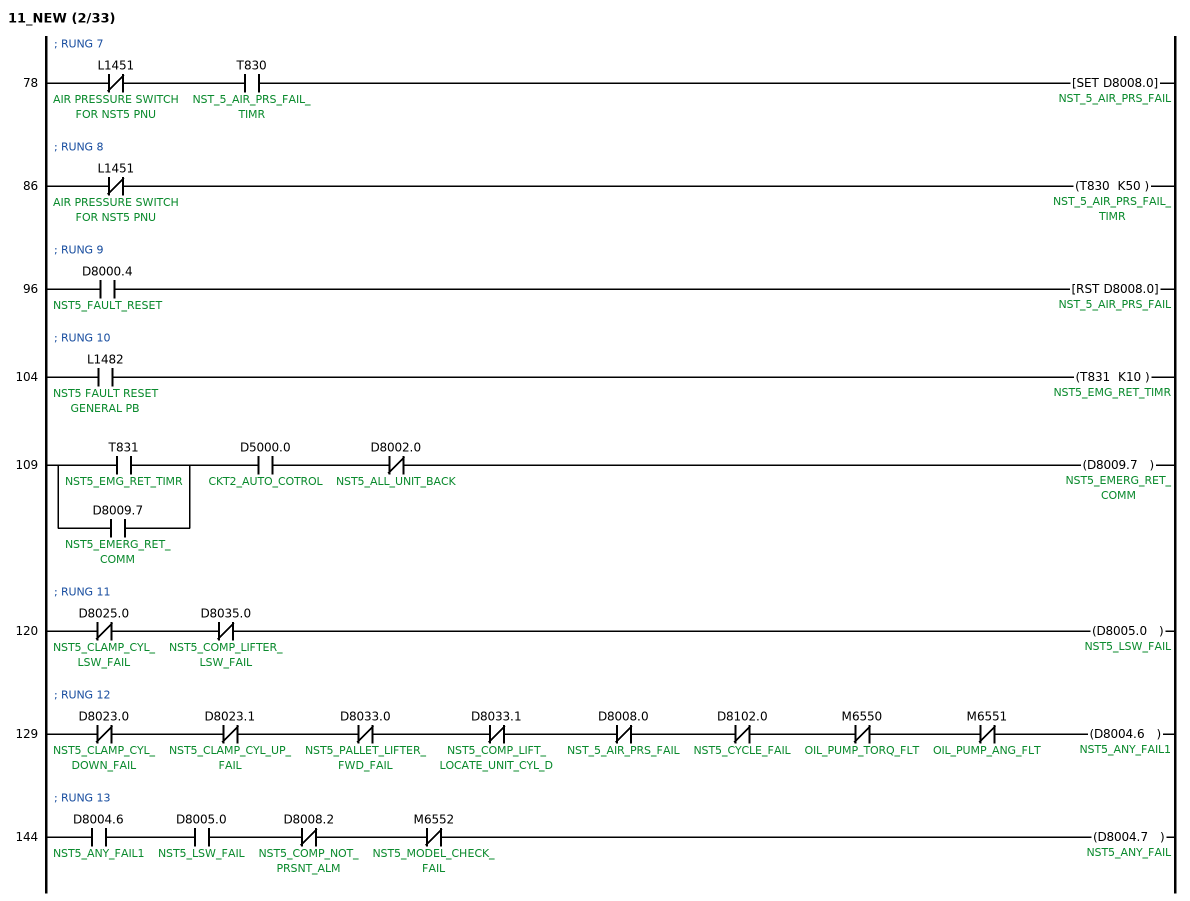
[picture p192: ladder of 11_NEW, rungs at steps 78 to 144]
; RUNG 7
78    LDI     L1451  ; AIR PRESSURE SWITCH FOR NST5 PNU
      AND     T830  ; NST_5_AIR_PRS_FAIL_TIMR
      SET     D8008.0  ; NST_5_AIR_PRS_FAIL
; RUNG 8
86    LDI     L1451  ; AIR PRESSURE SWITCH FOR NST5 PNU
      OUT     T830 K50  ; NST_5_AIR_PRS_FAIL_TIMR
; RUNG 9
96    LD      D8000.4  ; NST5_FAULT_RESET
      RST     D8008.0  ; NST_5_AIR_PRS_FAIL
; RUNG 10
104   LD      L1482  ; NST5 FAULT RESET GENERAL PB
      OUT     T831 K10  ; NST5_EMG_RET_TIMR
109   LD      T831  ; NST5_EMG_RET_TIMR
      OR      D8009.7  ; NST5_EMERG_RET_COMM
      AND     D5000.0  ; CKT2_AUTO_COTROL
      ANI     D8002.0  ; NST5_ALL_UNIT_BACK
      OUT     D8009.7  ; NST5_EMERG_RET_COMM
; RUNG 11
120   LDI     D8025.0  ; NST5_CLAMP_CYL_LSW_FAIL
      ANI     D8035.0  ; NST5_COMP_LIFTER_LSW_FAIL
      OUT     D8005.0  ; NST5_LSW_FAIL
; RUNG 12
129   LDI     D8023.0  ; NST5_CLAMP_CYL_DOWN_FAIL
      ANI     D8023.1  ; NST5_CLAMP_CYL_UP_FAIL
      ANI     D8033.0  ; NST5_PALLET_LIFTER_FWD_FAIL
      ANI     D8033.1  ; NST5_COMP_LIFT_LOCATE_UNIT_CYL_D
      ANI     D8008.0  ; NST_5_AIR_PRS_FAIL
      ANI     D8102.0  ; NST5_CYCLE_FAIL
      ANI     M6550  ; OIL_PUMP_TORQ_FLT
      ANI     M6551  ; OIL_PUMP_ANG_FLT
      OUT     D8004.6  ; NST5_ANY_FAIL1
; RUNG 13
144   LD      D8004.6  ; NST5_ANY_FAIL1
      AND     D8005.0  ; NST5_LSW_FAIL
      ANI     D8008.2  ; NST5_COMP_NOT_PRSNT_ALM
      ANI     M6552  ; NST5_MODEL_CHECK_FAIL
      OUT     D8004.7  ; NST5_ANY_FAIL
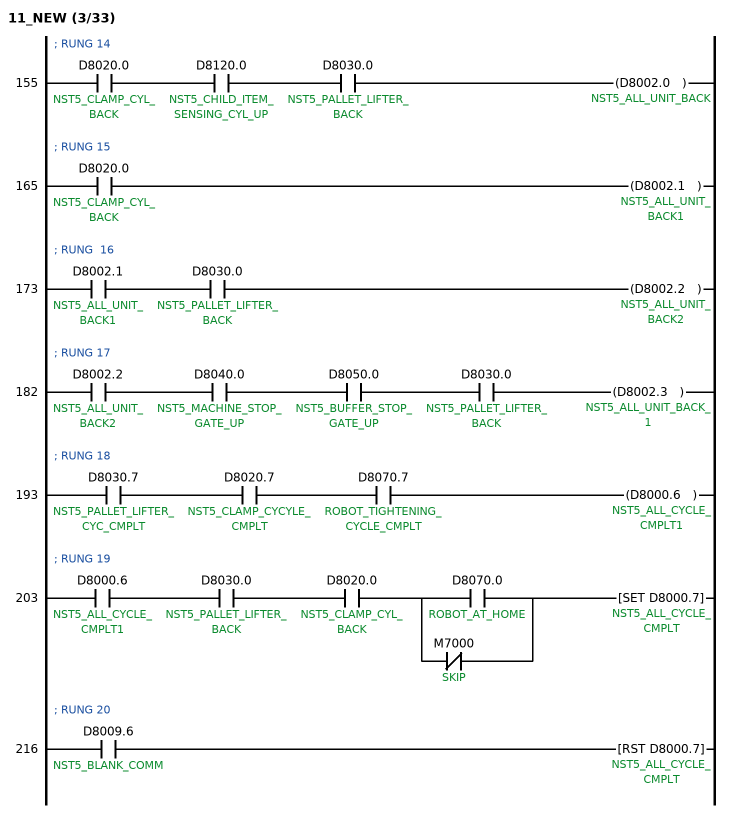
; RUNG 14
155   LD      D8020.0  ; NST5_CLAMP_CYL_BACK
      AND     D8120.0  ; NST5_CHILD_ITEM_SENSING_CYL_UP
      AND     D8030.0  ; NST5_PALLET_LIFTER_BACK
      OUT     D8002.0  ; NST5_ALL_UNIT_BACK
; RUNG 15
165   LD      D8020.0  ; NST5_CLAMP_CYL_BACK
      OUT     D8002.1  ; NST5_ALL_UNIT_BACK1
; RUNG  16
173   LD      D8002.1  ; NST5_ALL_UNIT_BACK1
      AND     D8030.0  ; NST5_PALLET_LIFTER_BACK
      OUT     D8002.2  ; NST5_ALL_UNIT_BACK2
; RUNG 17
182   LD      D8002.2  ; NST5_ALL_UNIT_BACK2
      AND     D8040.0  ; NST5_MACHINE_STOP_GATE_UP
      AND     D8050.0  ; NST5_BUFFER_STOP_GATE_UP
      AND     D8030.0  ; NST5_PALLET_LIFTER_BACK
      OUT     D8002.3  ; NST5_ALL_UNIT_BACK_1
; RUNG 18
193   LD      D8030.7  ; NST5_PALLET_LIFTER_CYC_CMPLT
      AND     D8020.7  ; NST5_CLAMP_CYCYLE_CMPLT
      AND     D8070.7  ; ROBOT_TIGHTENING_CYCLE_CMPLT
      OUT     D8000.6  ; NST5_ALL_CYCLE_CMPLT1
; RUNG 19
203   LD      D8000.6  ; NST5_ALL_CYCLE_CMPLT1
      AND     D8030.0  ; NST5_PALLET_LIFTER_BACK
      AND     D8020.0  ; NST5_CLAMP_CYL_BACK
      LD      D8070.0  ; ROBOT_AT_HOME
      ORI     M7000  ; SKIP
      ANB
      SET     D8000.7  ; NST5_ALL_CYCLE_CMPLT
; RUNG 20
216   LD      D8009.6  ; NST5_BLANK_COMM
      RST     D8000.7  ; NST5_ALL_CYCLE_CMPLT
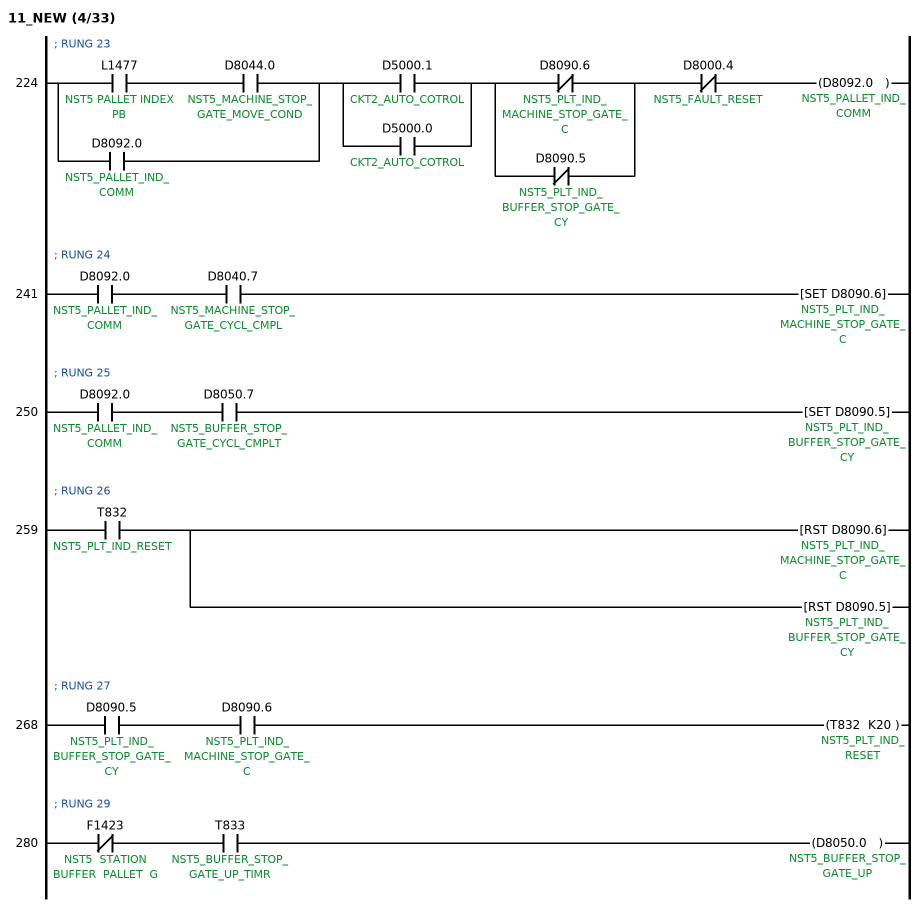
; RUNG 23
224   LD      L1477  ; NST5 PALLET INDEX PB
      AND     D8044.0  ; NST5_MACHINE_STOP_GATE_MOVE_COND
      OR      D8092.0  ; NST5_PALLET_IND_COMM
      LD      D5000.1  ; CKT2_AUTO_COTROL
      OR      D5000.0  ; CKT2_AUTO_COTROL
      ANB
      LDI     D8090.6  ; NST5_PLT_IND_MACHINE_STOP_GATE_C
      ORI     D8090.5  ; NST5_PLT_IND_BUFFER_STOP_GATE_CY
      ANB
      ANI     D8000.4  ; NST5_FAULT_RESET
      OUT     D8092.0  ; NST5_PALLET_IND_COMM
; RUNG 24
241   LD      D8092.0  ; NST5_PALLET_IND_COMM
      AND     D8040.7  ; NST5_MACHINE_STOP_GATE_CYCL_CMPL
      SET     D8090.6  ; NST5_PLT_IND_MACHINE_STOP_GATE_C
; RUNG 25
250   LD      D8092.0  ; NST5_PALLET_IND_COMM
      AND     D8050.7  ; NST5_BUFFER_STOP_GATE_CYCL_CMPLT
      SET     D8090.5  ; NST5_PLT_IND_BUFFER_STOP_GATE_CY
; RUNG 26
259   LD      T832  ; NST5_PLT_IND_RESET
      RST     D8090.6  ; NST5_PLT_IND_MACHINE_STOP_GATE_C
      RST     D8090.5  ; NST5_PLT_IND_BUFFER_STOP_GATE_CY
; RUNG 27
268   LD      D8090.5  ; NST5_PLT_IND_BUFFER_STOP_GATE_CY
      AND     D8090.6  ; NST5_PLT_IND_MACHINE_STOP_GATE_C
      OUT     T832 K20  ; NST5_PLT_IND_RESET
; RUNG 29
280   LDI     F1423  ; NST5  STATION  BUFFER  PALLET  G
      AND     T833  ; NST5_BUFFER_STOP_GATE_UP_TIMR
      OUT     D8050.0  ; NST5_BUFFER_STOP_GATE_UP
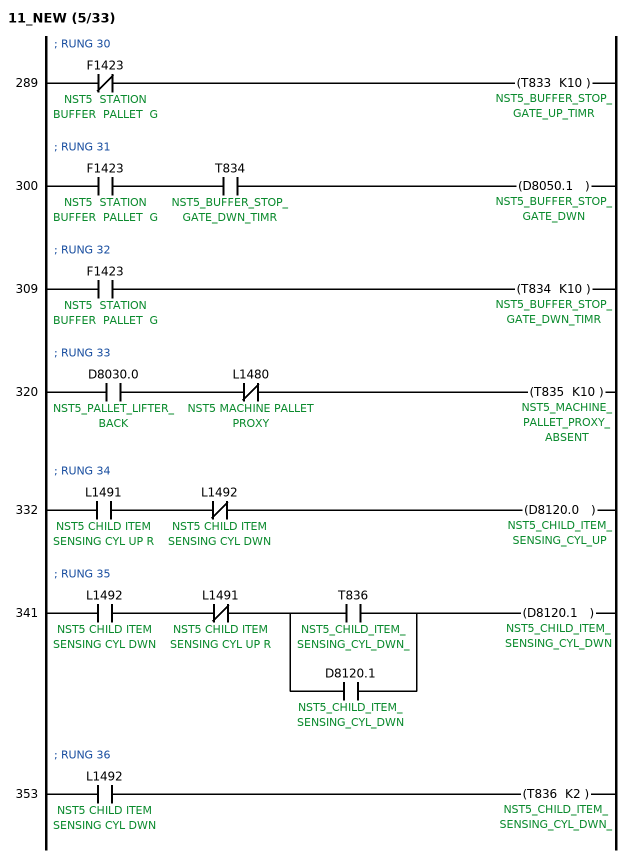
; RUNG 30
289   LDI     F1423  ; NST5  STATION  BUFFER  PALLET  G
      OUT     T833 K10  ; NST5_BUFFER_STOP_GATE_UP_TIMR
; RUNG 31
300   LD      F1423  ; NST5  STATION  BUFFER  PALLET  G
      AND     T834  ; NST5_BUFFER_STOP_GATE_DWN_TIMR
      OUT     D8050.1  ; NST5_BUFFER_STOP_GATE_DWN
; RUNG 32
309   LD      F1423  ; NST5  STATION  BUFFER  PALLET  G
      OUT     T834 K10  ; NST5_BUFFER_STOP_GATE_DWN_TIMR
; RUNG 33
320   LD      D8030.0  ; NST5_PALLET_LIFTER_BACK
      ANI     L1480  ; NST5 MACHINE PALLET PROXY
      OUT     T835 K10  ; NST5_MACHINE_PALLET_PROXY_ABSENT
; RUNG 34
332   LD      L1491  ; NST5 CHILD ITEM SENSING CYL UP R
      ANI     L1492  ; NST5 CHILD ITEM SENSING CYL DWN
      OUT     D8120.0  ; NST5_CHILD_ITEM_SENSING_CYL_UP
; RUNG 35
341   LD      L1492  ; NST5 CHILD ITEM SENSING CYL DWN
      ANI     L1491  ; NST5 CHILD ITEM SENSING CYL UP R
      LD      T836  ; NST5_CHILD_ITEM_SENSING_CYL_DWN_
      OR      D8120.1  ; NST5_CHILD_ITEM_SENSING_CYL_DWN
      ANB
      OUT     D8120.1  ; NST5_CHILD_ITEM_SENSING_CYL_DWN
; RUNG 36
353   LD      L1492  ; NST5 CHILD ITEM SENSING CYL DWN
      OUT     T836 K2  ; NST5_CHILD_ITEM_SENSING_CYL_DWN_
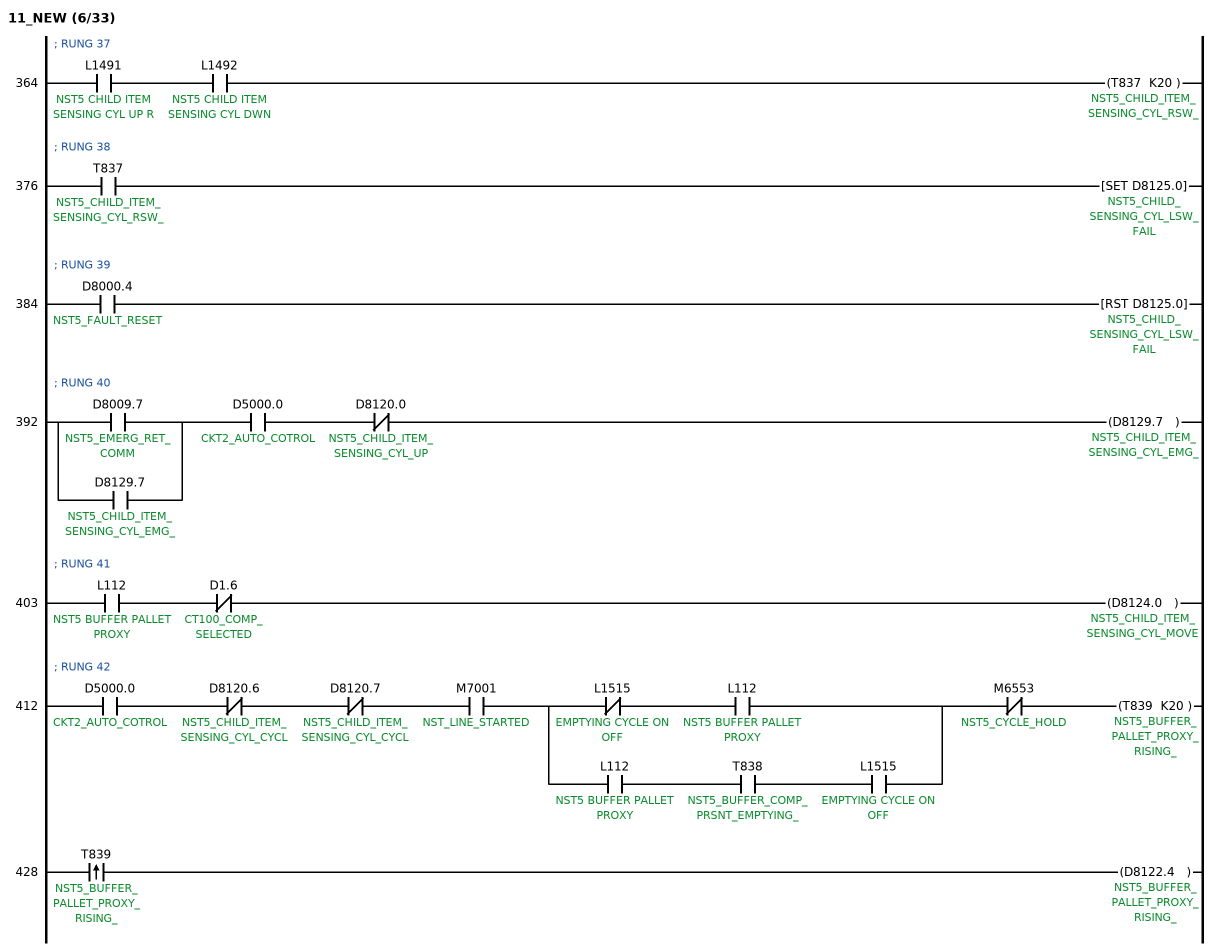
; RUNG 37
364   LD      L1491  ; NST5 CHILD ITEM SENSING CYL UP R
      AND     L1492  ; NST5 CHILD ITEM SENSING CYL DWN
      OUT     T837 K20  ; NST5_CHILD_ITEM_SENSING_CYL_RSW_
; RUNG 38
376   LD      T837  ; NST5_CHILD_ITEM_SENSING_CYL_RSW_
      SET     D8125.0  ; NST5_CHILD_SENSING_CYL_LSW_FAIL
; RUNG 39
384   LD      D8000.4  ; NST5_FAULT_RESET
      RST     D8125.0  ; NST5_CHILD_SENSING_CYL_LSW_FAIL
; RUNG 40
392   LD      D8009.7  ; NST5_EMERG_RET_COMM
      OR      D8129.7  ; NST5_CHILD_ITEM_SENSING_CYL_EMG_
      AND     D5000.0  ; CKT2_AUTO_COTROL
      ANI     D8120.0  ; NST5_CHILD_ITEM_SENSING_CYL_UP
      OUT     D8129.7  ; NST5_CHILD_ITEM_SENSING_CYL_EMG_
; RUNG 41
403   LD      L112  ; NST5 BUFFER PALLET PROXY
      ANI     D1.6  ; CT100_COMP_SELECTED
      OUT     D8124.0  ; NST5_CHILD_ITEM_SENSING_CYL_MOVE
; RUNG 42
412   LD      D5000.0  ; CKT2_AUTO_COTROL
      ANI     D8120.6  ; NST5_CHILD_ITEM_SENSING_CYL_CYCL
      ANI     D8120.7  ; NST5_CHILD_ITEM_SENSING_CYL_CYCL
      AND     M7001  ; NST_LINE_STARTED
      LDI     L1515  ; EMPTYING CYCLE ON OFF
      AND     L112  ; NST5 BUFFER PALLET PROXY
      LD      L112  ; NST5 BUFFER PALLET PROXY
      AND     T838  ; NST5_BUFFER_COMP_PRSNT_EMPTYING_
      AND     L1515  ; EMPTYING CYCLE ON OFF
      ORB
      ANB
      ANI     M6553  ; NST5_CYCLE_HOLD
      OUT     T839 K20  ; NST5_BUFFER_PALLET_PROXY_RISING_
428   LDP     T839  ; NST5_BUFFER_PALLET_PROXY_RISING_
      OUT     D8122.4  ; NST5_BUFFER_PALLET_PROXY_RISING_
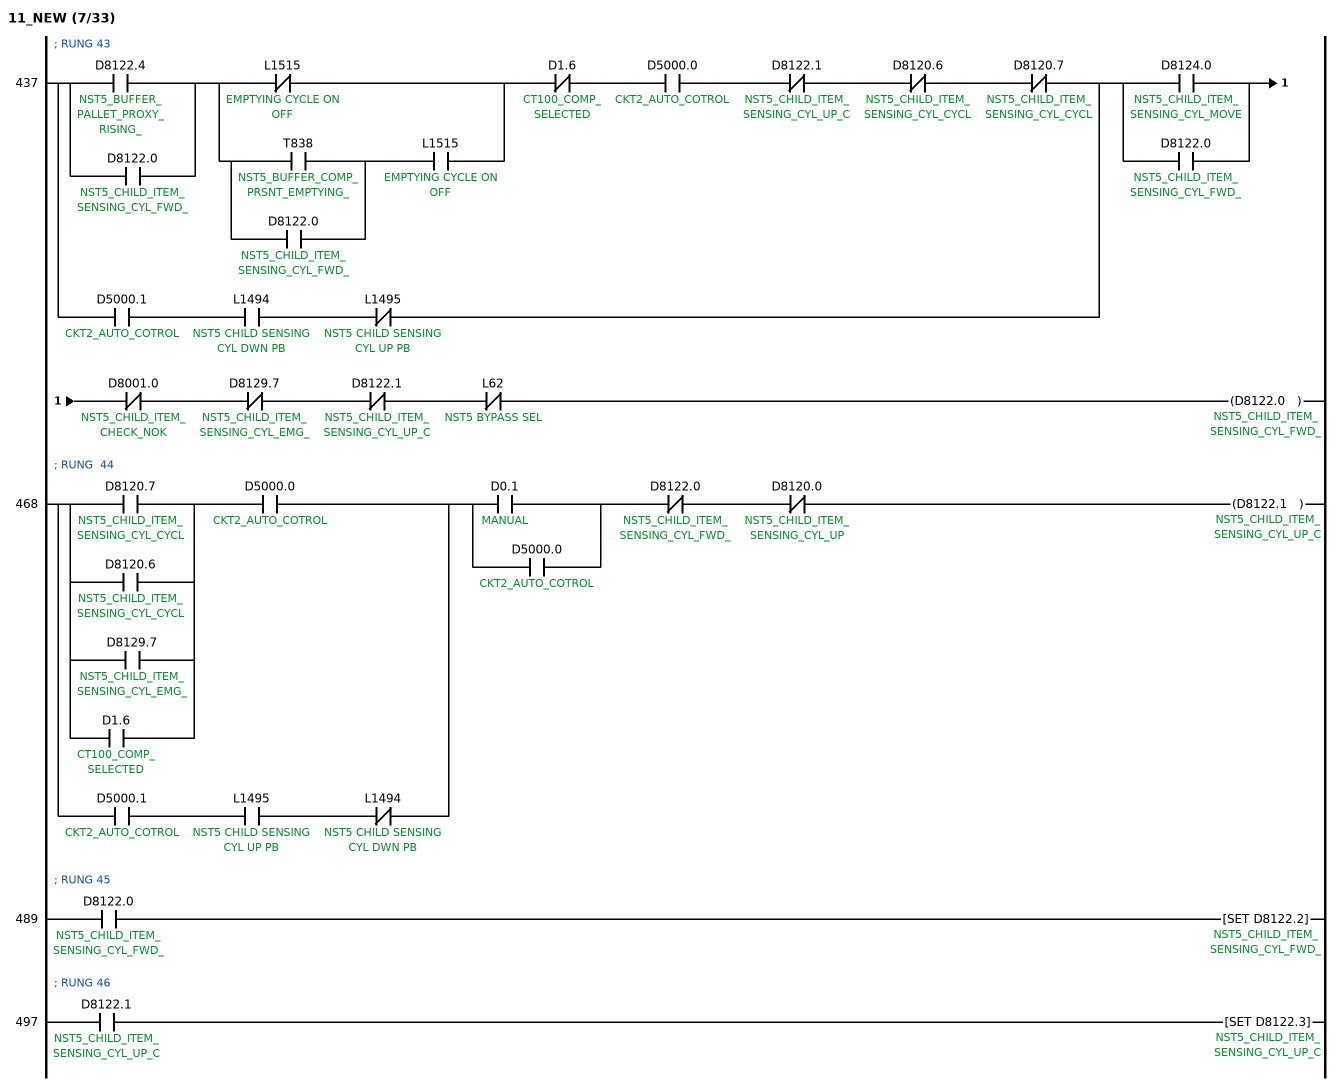
; RUNG 43
437   LD      D8122.4  ; NST5_BUFFER_PALLET_PROXY_RISING_
      OR      D8122.0  ; NST5_CHILD_ITEM_SENSING_CYL_FWD_
      LDI     L1515  ; EMPTYING CYCLE ON OFF
      LD      T838  ; NST5_BUFFER_COMP_PRSNT_EMPTYING_
      OR      D8122.0  ; NST5_CHILD_ITEM_SENSING_CYL_FWD_
      AND     L1515  ; EMPTYING CYCLE ON OFF
      ORB
      ANB
      ANI     D1.6  ; CT100_COMP_SELECTED
      AND     D5000.0  ; CKT2_AUTO_COTROL
      ANI     D8122.1  ; NST5_CHILD_ITEM_SENSING_CYL_UP_C
      ANI     D8120.6  ; NST5_CHILD_ITEM_SENSING_CYL_CYCL
      ANI     D8120.7  ; NST5_CHILD_ITEM_SENSING_CYL_CYCL
      LD      D5000.1  ; CKT2_AUTO_COTROL
      AND     L1494  ; NST5 CHILD SENSING CYL DWN PB
      ANI     L1495  ; NST5 CHILD SENSING CYL UP PB
      ORB
      LD      D8124.0  ; NST5_CHILD_ITEM_SENSING_CYL_MOVE
      OR      D8122.0  ; NST5_CHILD_ITEM_SENSING_CYL_FWD_
      ANB
      ANI     D8001.0  ; NST5_CHILD_ITEM_CHECK_NOK
      ANI     D8129.7  ; NST5_CHILD_ITEM_SENSING_CYL_EMG_
      ANI     D8122.1  ; NST5_CHILD_ITEM_SENSING_CYL_UP_C
      ANI     L62  ; NST5 BYPASS SEL
      OUT     D8122.0  ; NST5_CHILD_ITEM_SENSING_CYL_FWD_
; RUNG  44
468   LD      D8120.7  ; NST5_CHILD_ITEM_SENSING_CYL_CYCL
      OR      D8120.6  ; NST5_CHILD_ITEM_SENSING_CYL_CYCL
      OR      D8129.7  ; NST5_CHILD_ITEM_SENSING_CYL_EMG_
      OR      D1.6  ; CT100_COMP_SELECTED
      AND     D5000.0  ; CKT2_AUTO_COTROL
      LD      D5000.1  ; CKT2_AUTO_COTROL
      AND     L1495  ; NST5 CHILD SENSING CYL UP PB
      ANI     L1494  ; NST5 CHILD SENSING CYL DWN PB
      ORB
      LD      D0.1  ; MANUAL
      OR      D5000.0  ; CKT2_AUTO_COTROL
      ANB
      ANI     D8122.0  ; NST5_CHILD_ITEM_SENSING_CYL_FWD_
      ANI     D8120.0  ; NST5_CHILD_ITEM_SENSING_CYL_UP
      OUT     D8122.1  ; NST5_CHILD_ITEM_SENSING_CYL_UP_C
; RUNG 45
489   LD      D8122.0  ; NST5_CHILD_ITEM_SENSING_CYL_FWD_
      SET     D8122.2  ; NST5_CHILD_ITEM_SENSING_CYL_FWD_
; RUNG 46
497   LD      D8122.1  ; NST5_CHILD_ITEM_SENSING_CYL_UP_C
      SET     D8122.3  ; NST5_CHILD_ITEM_SENSING_CYL_UP_C
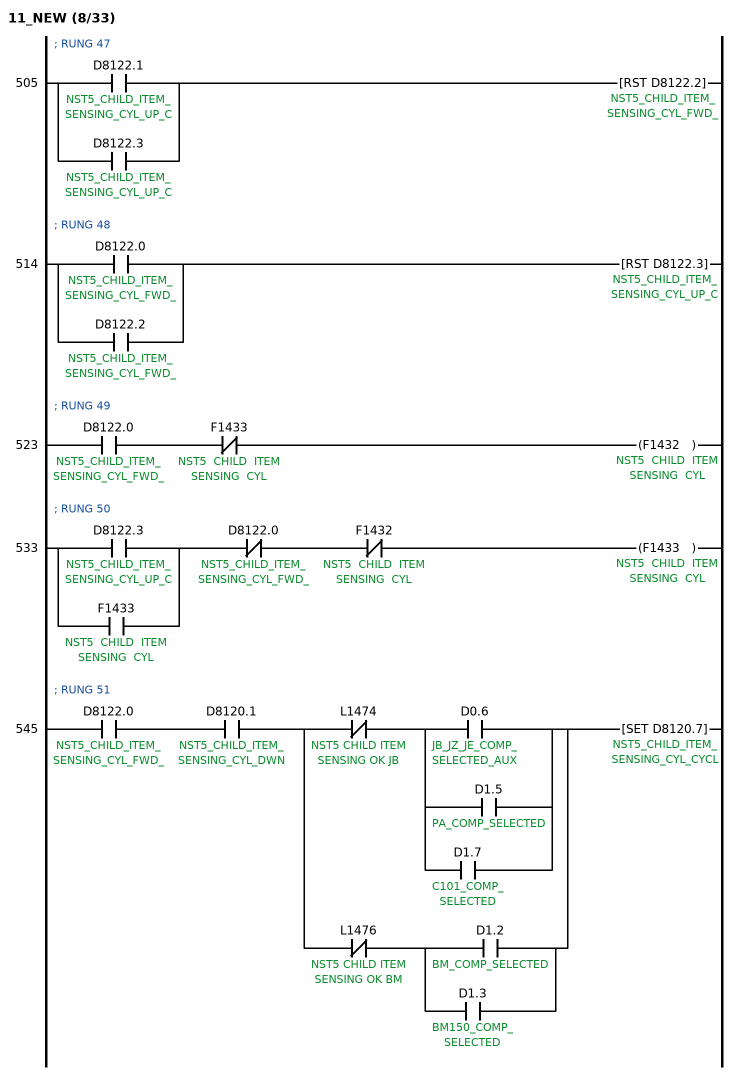
; RUNG 47
505   LD      D8122.1  ; NST5_CHILD_ITEM_SENSING_CYL_UP_C
      OR      D8122.3  ; NST5_CHILD_ITEM_SENSING_CYL_UP_C
      RST     D8122.2  ; NST5_CHILD_ITEM_SENSING_CYL_FWD_
; RUNG 48
514   LD      D8122.0  ; NST5_CHILD_ITEM_SENSING_CYL_FWD_
      OR      D8122.2  ; NST5_CHILD_ITEM_SENSING_CYL_FWD_
      RST     D8122.3  ; NST5_CHILD_ITEM_SENSING_CYL_UP_C
; RUNG 49
523   LD      D8122.0  ; NST5_CHILD_ITEM_SENSING_CYL_FWD_
      ANI     F1433  ; NST5  CHILD  ITEM  SENSING  CYL
      OUT     F1432  ; NST5  CHILD  ITEM  SENSING  CYL
; RUNG 50
533   LD      D8122.3  ; NST5_CHILD_ITEM_SENSING_CYL_UP_C
      OR      F1433  ; NST5  CHILD  ITEM  SENSING  CYL
      ANI     D8122.0  ; NST5_CHILD_ITEM_SENSING_CYL_FWD_
      ANI     F1432  ; NST5  CHILD  ITEM  SENSING  CYL
      OUT     F1433  ; NST5  CHILD  ITEM  SENSING  CYL
; RUNG 51
545   LD      D8122.0  ; NST5_CHILD_ITEM_SENSING_CYL_FWD_
      AND     D8120.1  ; NST5_CHILD_ITEM_SENSING_CYL_DWN
      LDI     L1474  ; NST5 CHILD ITEM SENSING OK JB
      LD      D0.6  ; JB_JZ_JE_COMP_SELECTED_AUX
      OR      D1.5  ; PA_COMP_SELECTED
      OR      D1.7  ; C101_COMP_SELECTED
      ANB
      LDI     L1476  ; NST5 CHILD ITEM SENSING OK BM
      LD      D1.2  ; BM_COMP_SELECTED
      OR      D1.3  ; BM150_COMP_SELECTED
      ANB
      ORB
      ANB
      SET     D8120.7  ; NST5_CHILD_ITEM_SENSING_CYL_CYCL
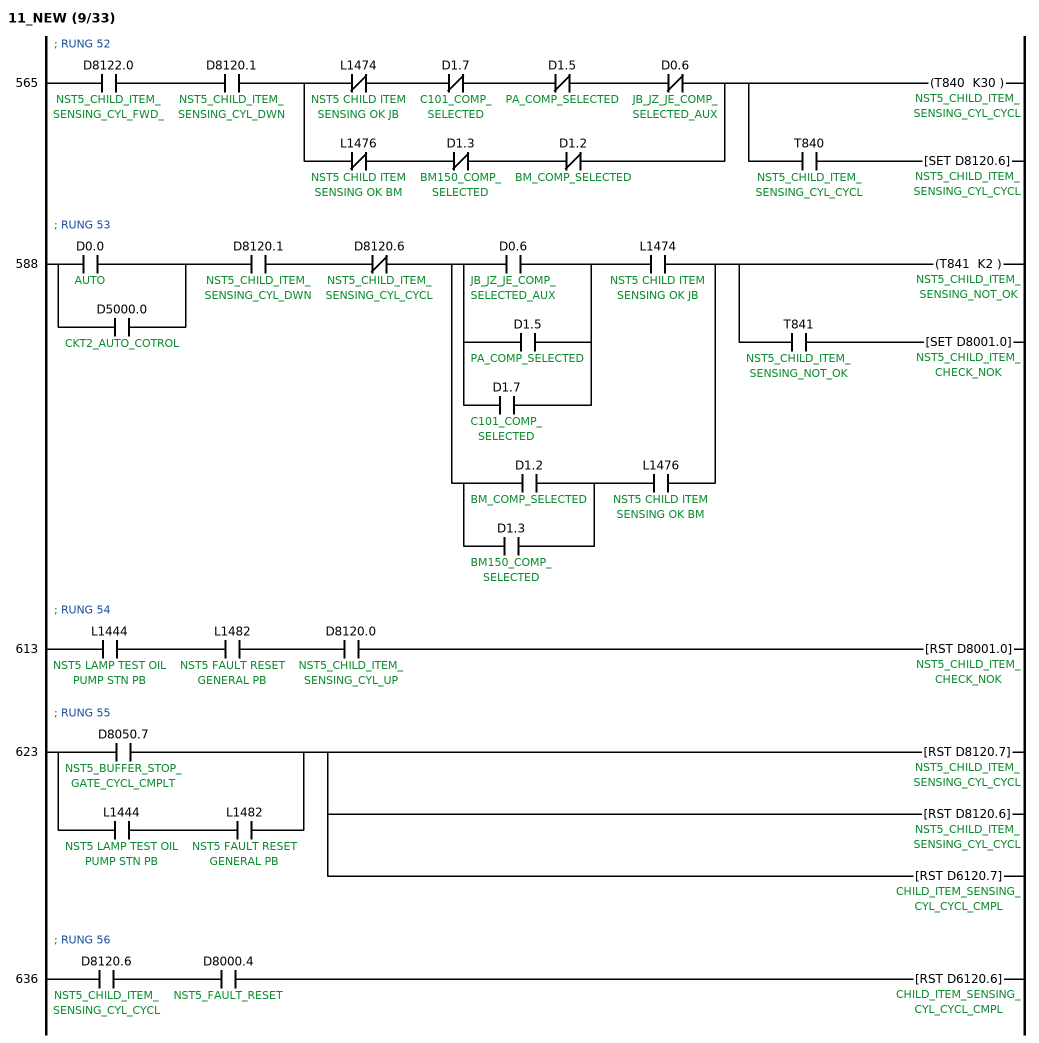
; RUNG 52
565   LD      D8122.0  ; NST5_CHILD_ITEM_SENSING_CYL_FWD_
      AND     D8120.1  ; NST5_CHILD_ITEM_SENSING_CYL_DWN
      LDI     L1474  ; NST5 CHILD ITEM SENSING OK JB
      ANI     D1.7  ; C101_COMP_SELECTED
      ANI     D1.5  ; PA_COMP_SELECTED
      ANI     D0.6  ; JB_JZ_JE_COMP_SELECTED_AUX
      LDI     L1476  ; NST5 CHILD ITEM SENSING OK BM
      ANI     D1.3  ; BM150_COMP_SELECTED
      ANI     D1.2  ; BM_COMP_SELECTED
      ORB
      ANB
      OUT     T840 K30  ; NST5_CHILD_ITEM_SENSING_CYL_CYCL
      AND     T840  ; NST5_CHILD_ITEM_SENSING_CYL_CYCL
      SET     D8120.6  ; NST5_CHILD_ITEM_SENSING_CYL_CYCL
; RUNG 53
588   LD      D0.0  ; AUTO
      OR      D5000.0  ; CKT2_AUTO_COTROL
      AND     D8120.1  ; NST5_CHILD_ITEM_SENSING_CYL_DWN
      ANI     D8120.6  ; NST5_CHILD_ITEM_SENSING_CYL_CYCL
      LD      D0.6  ; JB_JZ_JE_COMP_SELECTED_AUX
      OR      D1.5  ; PA_COMP_SELECTED
      OR      D1.7  ; C101_COMP_SELECTED
      AND     L1474  ; NST5 CHILD ITEM SENSING OK JB
      LD      D1.2  ; BM_COMP_SELECTED
      OR      D1.3  ; BM150_COMP_SELECTED
      AND     L1476  ; NST5 CHILD ITEM SENSING OK BM
      ORB
      ANB
      OUT     T841 K2  ; NST5_CHILD_ITEM_SENSING_NOT_OK
      AND     T841  ; NST5_CHILD_ITEM_SENSING_NOT_OK
      SET     D8001.0  ; NST5_CHILD_ITEM_CHECK_NOK
; RUNG 54
613   LD      L1444  ; NST5 LAMP TEST OIL PUMP STN PB
      AND     L1482  ; NST5 FAULT RESET GENERAL PB
      AND     D8120.0  ; NST5_CHILD_ITEM_SENSING_CYL_UP
      RST     D8001.0  ; NST5_CHILD_ITEM_CHECK_NOK
; RUNG 55
623   LD      D8050.7  ; NST5_BUFFER_STOP_GATE_CYCL_CMPLT
      LD      L1444  ; NST5 LAMP TEST OIL PUMP STN PB
      AND     L1482  ; NST5 FAULT RESET GENERAL PB
      ORB
      RST     D8120.7  ; NST5_CHILD_ITEM_SENSING_CYL_CYCL
      RST     D8120.6  ; NST5_CHILD_ITEM_SENSING_CYL_CYCL
      RST     D6120.7  ; CHILD_ITEM_SENSING_CYL_CYCL_CMPL
; RUNG 56
636   LD      D8120.6  ; NST5_CHILD_ITEM_SENSING_CYL_CYCL
      AND     D8000.4  ; NST5_FAULT_RESET
      RST     D6120.6  ; CHILD_ITEM_SENSING_CYL_CYCL_CMPL
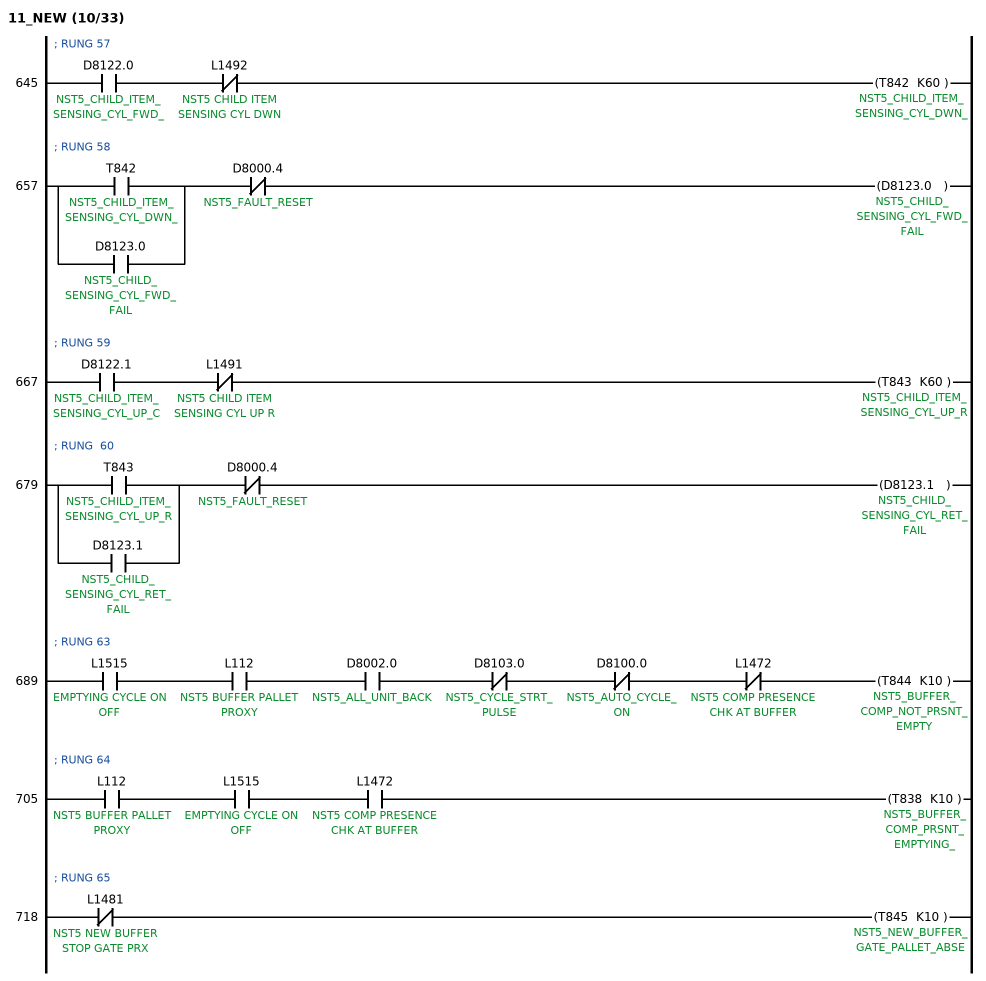
; RUNG 57
645   LD      D8122.0  ; NST5_CHILD_ITEM_SENSING_CYL_FWD_
      ANI     L1492  ; NST5 CHILD ITEM SENSING CYL DWN
      OUT     T842 K60  ; NST5_CHILD_ITEM_SENSING_CYL_DWN_
; RUNG 58
657   LD      T842  ; NST5_CHILD_ITEM_SENSING_CYL_DWN_
      OR      D8123.0  ; NST5_CHILD_SENSING_CYL_FWD_FAIL
      ANI     D8000.4  ; NST5_FAULT_RESET
      OUT     D8123.0  ; NST5_CHILD_SENSING_CYL_FWD_FAIL
; RUNG 59
667   LD      D8122.1  ; NST5_CHILD_ITEM_SENSING_CYL_UP_C
      ANI     L1491  ; NST5 CHILD ITEM SENSING CYL UP R
      OUT     T843 K60  ; NST5_CHILD_ITEM_SENSING_CYL_UP_R
; RUNG  60
679   LD      T843  ; NST5_CHILD_ITEM_SENSING_CYL_UP_R
      OR      D8123.1  ; NST5_CHILD_SENSING_CYL_RET_FAIL
      ANI     D8000.4  ; NST5_FAULT_RESET
      OUT     D8123.1  ; NST5_CHILD_SENSING_CYL_RET_FAIL
; RUNG 63
689   LD      L1515  ; EMPTYING CYCLE ON OFF
      AND     L112  ; NST5 BUFFER PALLET PROXY
      AND     D8002.0  ; NST5_ALL_UNIT_BACK
      ANI     D8103.0  ; NST5_CYCLE_STRT_PULSE
      ANI     D8100.0  ; NST5_AUTO_CYCLE_ON
      ANI     L1472  ; NST5 COMP PRESENCE CHK AT BUFFER
      OUT     T844 K10  ; NST5_BUFFER_COMP_NOT_PRSNT_EMPTY
; RUNG 64
705   LD      L112  ; NST5 BUFFER PALLET PROXY
      AND     L1515  ; EMPTYING CYCLE ON OFF
      AND     L1472  ; NST5 COMP PRESENCE CHK AT BUFFER
      OUT     T838 K10  ; NST5_BUFFER_COMP_PRSNT_EMPTYING_
; RUNG 65
718   LDI     L1481  ; NST5 NEW BUFFER STOP GATE PRX
      OUT     T845 K10  ; NST5_NEW_BUFFER_GATE_PALLET_ABSE
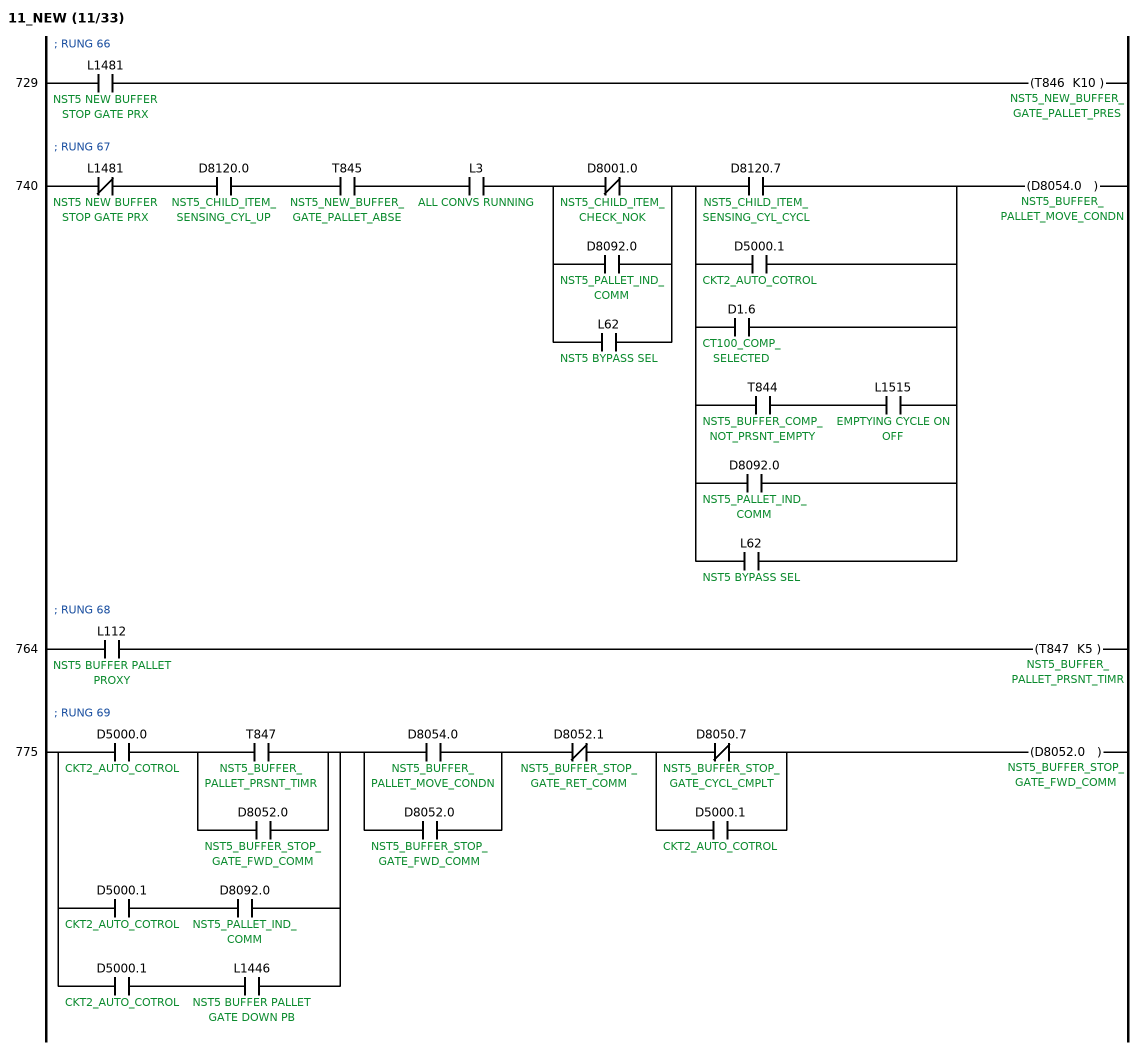
; RUNG 66
729   LD      L1481  ; NST5 NEW BUFFER STOP GATE PRX
      OUT     T846 K10  ; NST5_NEW_BUFFER_GATE_PALLET_PRES
; RUNG 67
740   LDI     L1481  ; NST5 NEW BUFFER STOP GATE PRX
      AND     D8120.0  ; NST5_CHILD_ITEM_SENSING_CYL_UP
      AND     T845  ; NST5_NEW_BUFFER_GATE_PALLET_ABSE
      AND     L3  ; ALL CONVS RUNNING
      LDI     D8001.0  ; NST5_CHILD_ITEM_CHECK_NOK
      OR      D8092.0  ; NST5_PALLET_IND_COMM
      OR      L62  ; NST5 BYPASS SEL
      ANB
      LD      D8120.7  ; NST5_CHILD_ITEM_SENSING_CYL_CYCL
      OR      D5000.1  ; CKT2_AUTO_COTROL
      OR      D1.6  ; CT100_COMP_SELECTED
      LD      T844  ; NST5_BUFFER_COMP_NOT_PRSNT_EMPTY
      AND     L1515  ; EMPTYING CYCLE ON OFF
      ORB
      OR      D8092.0  ; NST5_PALLET_IND_COMM
      OR      L62  ; NST5 BYPASS SEL
      ANB
      OUT     D8054.0  ; NST5_BUFFER_PALLET_MOVE_CONDN
; RUNG 68
764   LD      L112  ; NST5 BUFFER PALLET PROXY
      OUT     T847 K5  ; NST5_BUFFER_PALLET_PRSNT_TIMR
; RUNG 69
775   LD      D5000.0  ; CKT2_AUTO_COTROL
      LD      T847  ; NST5_BUFFER_PALLET_PRSNT_TIMR
      OR      D8052.0  ; NST5_BUFFER_STOP_GATE_FWD_COMM
      ANB
      LD      D5000.1  ; CKT2_AUTO_COTROL
      AND     D8092.0  ; NST5_PALLET_IND_COMM
      ORB
      LD      D5000.1  ; CKT2_AUTO_COTROL
      AND     L1446  ; NST5 BUFFER PALLET GATE DOWN PB
      ORB
      LD      D8054.0  ; NST5_BUFFER_PALLET_MOVE_CONDN
      OR      D8052.0  ; NST5_BUFFER_STOP_GATE_FWD_COMM
      ANB
      ANI     D8052.1  ; NST5_BUFFER_STOP_GATE_RET_COMM
      LDI     D8050.7  ; NST5_BUFFER_STOP_GATE_CYCL_CMPLT
      OR      D5000.1  ; CKT2_AUTO_COTROL
      ANB
      OUT     D8052.0  ; NST5_BUFFER_STOP_GATE_FWD_COMM
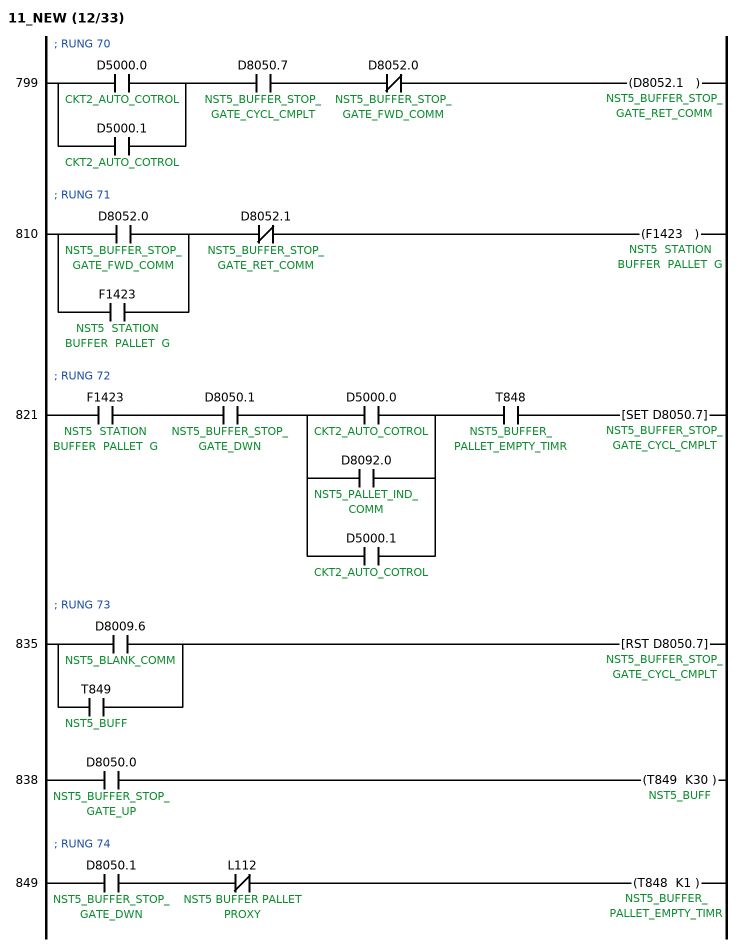
; RUNG 70
799   LD      D5000.0  ; CKT2_AUTO_COTROL
      OR      D5000.1  ; CKT2_AUTO_COTROL
      AND     D8050.7  ; NST5_BUFFER_STOP_GATE_CYCL_CMPLT
      ANI     D8052.0  ; NST5_BUFFER_STOP_GATE_FWD_COMM
      OUT     D8052.1  ; NST5_BUFFER_STOP_GATE_RET_COMM
; RUNG 71
810   LD      D8052.0  ; NST5_BUFFER_STOP_GATE_FWD_COMM
      OR      F1423  ; NST5  STATION  BUFFER  PALLET  G
      ANI     D8052.1  ; NST5_BUFFER_STOP_GATE_RET_COMM
      OUT     F1423  ; NST5  STATION  BUFFER  PALLET  G
; RUNG 72
821   LD      F1423  ; NST5  STATION  BUFFER  PALLET  G
      AND     D8050.1  ; NST5_BUFFER_STOP_GATE_DWN
      LD      D5000.0  ; CKT2_AUTO_COTROL
      OR      D8092.0  ; NST5_PALLET_IND_COMM
      OR      D5000.1  ; CKT2_AUTO_COTROL
      ANB
      AND     T848  ; NST5_BUFFER_PALLET_EMPTY_TIMR
      SET     D8050.7  ; NST5_BUFFER_STOP_GATE_CYCL_CMPLT
; RUNG 73
835   LD      D8009.6  ; NST5_BLANK_COMM
      OR      T849  ; NST5_BUFF
      RST     D8050.7  ; NST5_BUFFER_STOP_GATE_CYCL_CMPLT
838   LD      D8050.0  ; NST5_BUFFER_STOP_GATE_UP
      OUT     T849 K30  ; NST5_BUFF
; RUNG 74
849   LD      D8050.1  ; NST5_BUFFER_STOP_GATE_DWN
      ANI     L112  ; NST5 BUFFER PALLET PROXY
      OUT     T848 K1  ; NST5_BUFFER_PALLET_EMPTY_TIMR
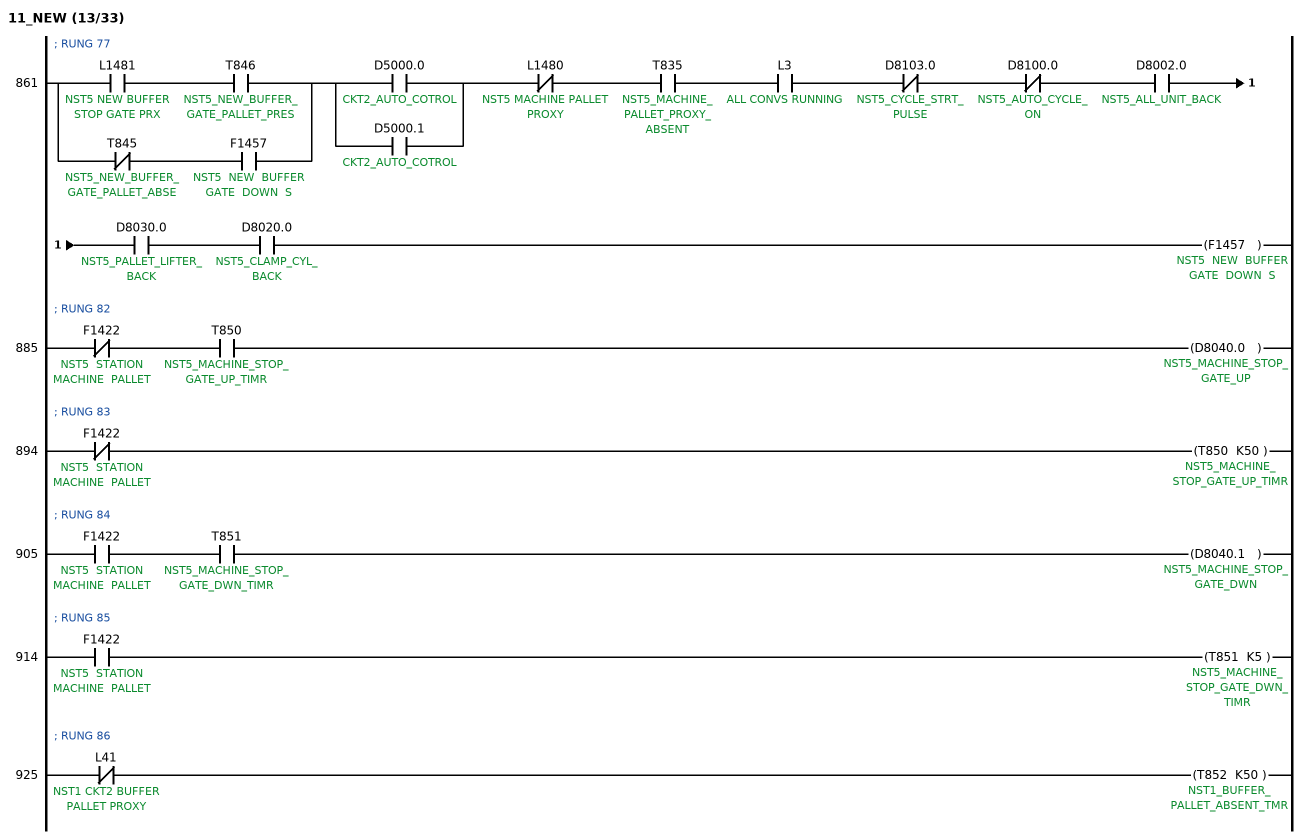
; RUNG 77
861   LD      L1481  ; NST5 NEW BUFFER STOP GATE PRX
      AND     T846  ; NST5_NEW_BUFFER_GATE_PALLET_PRES
      LDI     T845  ; NST5_NEW_BUFFER_GATE_PALLET_ABSE
      AND     F1457  ; NST5  NEW  BUFFER  GATE  DOWN  S
      ORB
      LD      D5000.0  ; CKT2_AUTO_COTROL
      OR      D5000.1  ; CKT2_AUTO_COTROL
      ANB
      ANI     L1480  ; NST5 MACHINE PALLET PROXY
      AND     T835  ; NST5_MACHINE_PALLET_PROXY_ABSENT
      AND     L3  ; ALL CONVS RUNNING
      ANI     D8103.0  ; NST5_CYCLE_STRT_PULSE
      ANI     D8100.0  ; NST5_AUTO_CYCLE_ON
      AND     D8002.0  ; NST5_ALL_UNIT_BACK
      AND     D8030.0  ; NST5_PALLET_LIFTER_BACK
      AND     D8020.0  ; NST5_CLAMP_CYL_BACK
      OUT     F1457  ; NST5  NEW  BUFFER  GATE  DOWN  S
; RUNG 82
885   LDI     F1422  ; NST5  STATION  MACHINE  PALLET
      AND     T850  ; NST5_MACHINE_STOP_GATE_UP_TIMR
      OUT     D8040.0  ; NST5_MACHINE_STOP_GATE_UP
; RUNG 83
894   LDI     F1422  ; NST5  STATION  MACHINE  PALLET
      OUT     T850 K50  ; NST5_MACHINE_STOP_GATE_UP_TIMR
; RUNG 84
905   LD      F1422  ; NST5  STATION  MACHINE  PALLET
      AND     T851  ; NST5_MACHINE_STOP_GATE_DWN_TIMR
      OUT     D8040.1  ; NST5_MACHINE_STOP_GATE_DWN
; RUNG 85
914   LD      F1422  ; NST5  STATION  MACHINE  PALLET
      OUT     T851 K5  ; NST5_MACHINE_STOP_GATE_DWN_TIMR
; RUNG 86
925   LDI     L41  ; NST1 CKT2 BUFFER PALLET PROXY
      OUT     T852 K50  ; NST1_BUFFER_PALLET_ABSENT_TMR
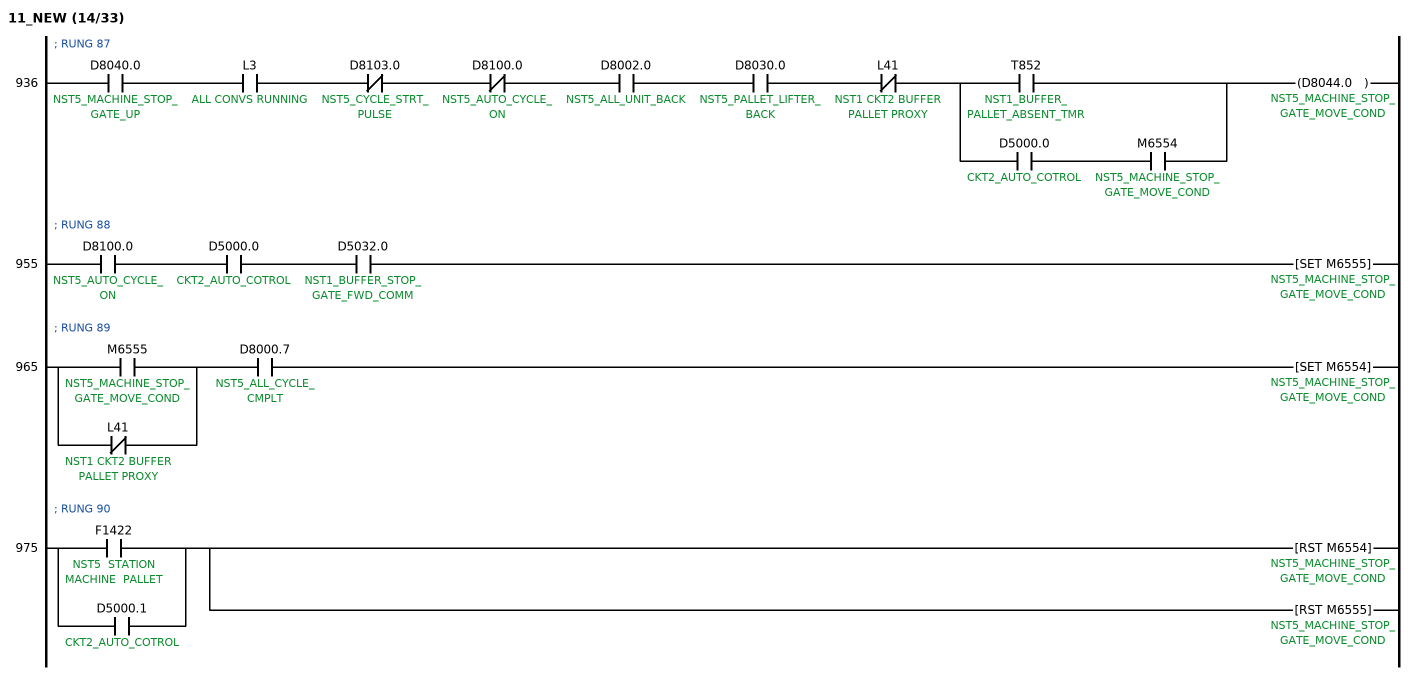
; RUNG 87
936   LD      D8040.0  ; NST5_MACHINE_STOP_GATE_UP
      AND     L3  ; ALL CONVS RUNNING
      ANI     D8103.0  ; NST5_CYCLE_STRT_PULSE
      ANI     D8100.0  ; NST5_AUTO_CYCLE_ON
      AND     D8002.0  ; NST5_ALL_UNIT_BACK
      AND     D8030.0  ; NST5_PALLET_LIFTER_BACK
      ANI     L41  ; NST1 CKT2 BUFFER PALLET PROXY
      LD      T852  ; NST1_BUFFER_PALLET_ABSENT_TMR
      LD      D5000.0  ; CKT2_AUTO_COTROL
      AND     M6554  ; NST5_MACHINE_STOP_GATE_MOVE_COND
      ORB
      ANB
      OUT     D8044.0  ; NST5_MACHINE_STOP_GATE_MOVE_COND
; RUNG 88
955   LD      D8100.0  ; NST5_AUTO_CYCLE_ON
      AND     D5000.0  ; CKT2_AUTO_COTROL
      AND     D5032.0  ; NST1_BUFFER_STOP_GATE_FWD_COMM
      SET     M6555  ; NST5_MACHINE_STOP_GATE_MOVE_COND
; RUNG 89
965   LD      M6555  ; NST5_MACHINE_STOP_GATE_MOVE_COND
      ORI     L41  ; NST1 CKT2 BUFFER PALLET PROXY
      AND     D8000.7  ; NST5_ALL_CYCLE_CMPLT
      SET     M6554  ; NST5_MACHINE_STOP_GATE_MOVE_COND
; RUNG 90
975   LD      F1422  ; NST5  STATION  MACHINE  PALLET
      OR      D5000.1  ; CKT2_AUTO_COTROL
      RST     M6554  ; NST5_MACHINE_STOP_GATE_MOVE_COND
      RST     M6555  ; NST5_MACHINE_STOP_GATE_MOVE_COND
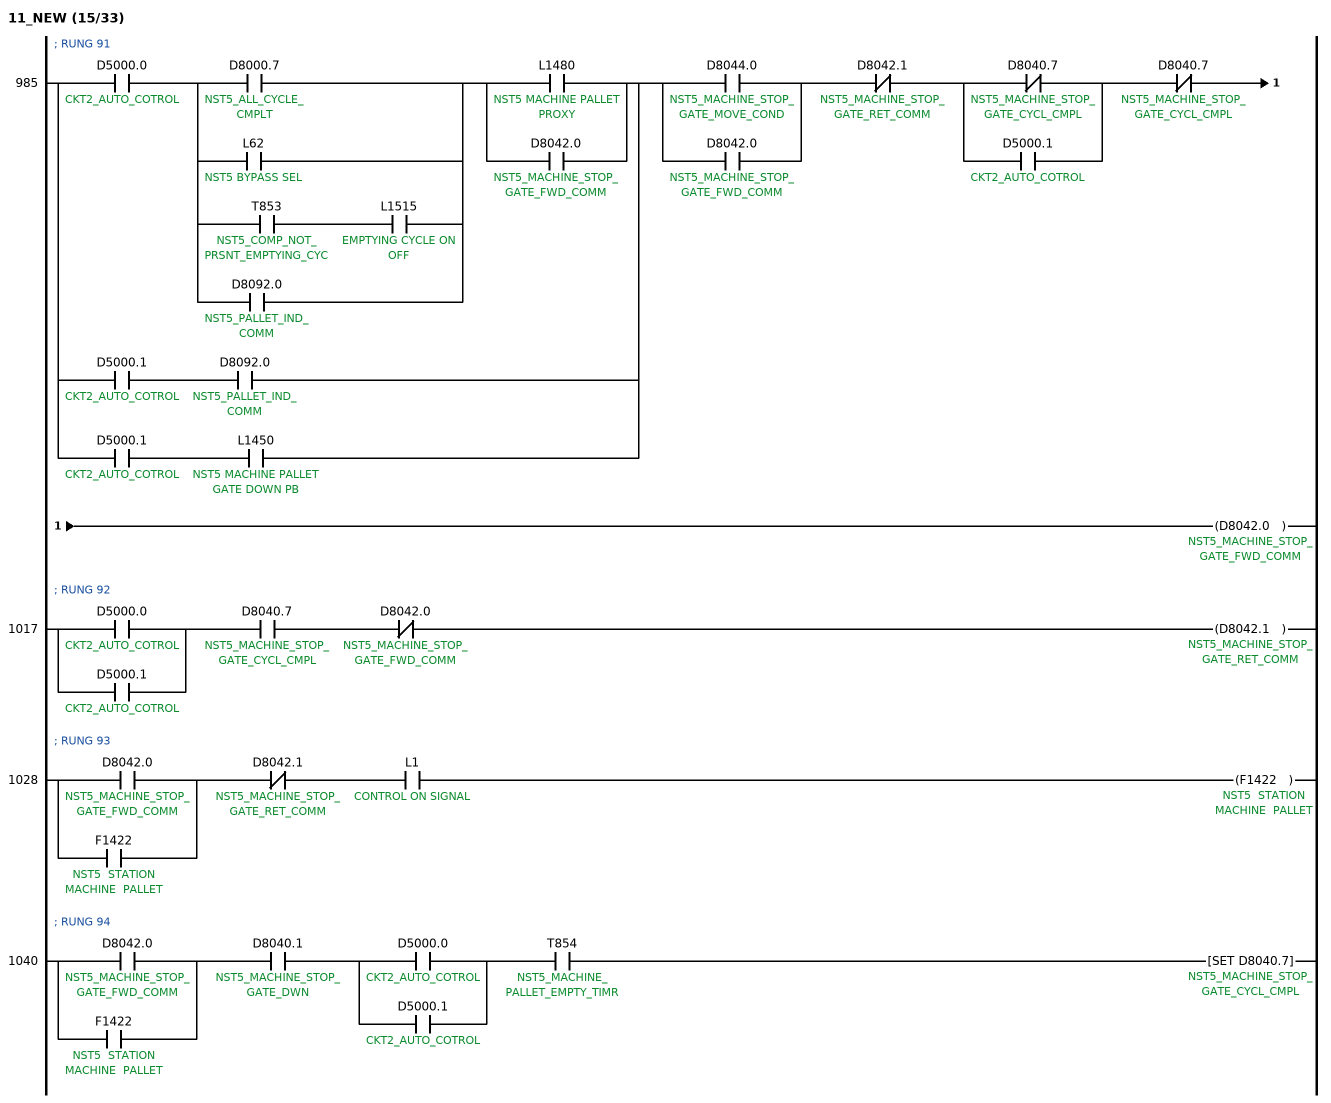
; RUNG 91
985   LD      D5000.0  ; CKT2_AUTO_COTROL
      LD      D8000.7  ; NST5_ALL_CYCLE_CMPLT
      OR      L62  ; NST5 BYPASS SEL
      LD      T853  ; NST5_COMP_NOT_PRSNT_EMPTYING_CYC
      AND     L1515  ; EMPTYING CYCLE ON OFF
      ORB
      OR      D8092.0  ; NST5_PALLET_IND_COMM
      ANB
      LD      L1480  ; NST5 MACHINE PALLET PROXY
      OR      D8042.0  ; NST5_MACHINE_STOP_GATE_FWD_COMM
      ANB
      LD      D5000.1  ; CKT2_AUTO_COTROL
      AND     D8092.0  ; NST5_PALLET_IND_COMM
      ORB
      LD      D5000.1  ; CKT2_AUTO_COTROL
      AND     L1450  ; NST5 MACHINE PALLET GATE DOWN PB
      ORB
      LD      D8044.0  ; NST5_MACHINE_STOP_GATE_MOVE_COND
      OR      D8042.0  ; NST5_MACHINE_STOP_GATE_FWD_COMM
      ANB
      ANI     D8042.1  ; NST5_MACHINE_STOP_GATE_RET_COMM
      LDI     D8040.7  ; NST5_MACHINE_STOP_GATE_CYCL_CMPL
      OR      D5000.1  ; CKT2_AUTO_COTROL
      ANB
      ANI     D8040.7  ; NST5_MACHINE_STOP_GATE_CYCL_CMPL
      OUT     D8042.0  ; NST5_MACHINE_STOP_GATE_FWD_COMM
; RUNG 92
1017  LD      D5000.0  ; CKT2_AUTO_COTROL
      OR      D5000.1  ; CKT2_AUTO_COTROL
      AND     D8040.7  ; NST5_MACHINE_STOP_GATE_CYCL_CMPL
      ANI     D8042.0  ; NST5_MACHINE_STOP_GATE_FWD_COMM
      OUT     D8042.1  ; NST5_MACHINE_STOP_GATE_RET_COMM
; RUNG 93
1028  LD      D8042.0  ; NST5_MACHINE_STOP_GATE_FWD_COMM
      OR      F1422  ; NST5  STATION  MACHINE  PALLET
      ANI     D8042.1  ; NST5_MACHINE_STOP_GATE_RET_COMM
      AND     L1  ; CONTROL ON SIGNAL
      OUT     F1422  ; NST5  STATION  MACHINE  PALLET
; RUNG 94
1040  LD      D8042.0  ; NST5_MACHINE_STOP_GATE_FWD_COMM
      OR      F1422  ; NST5  STATION  MACHINE  PALLET
      AND     D8040.1  ; NST5_MACHINE_STOP_GATE_DWN
      LD      D5000.0  ; CKT2_AUTO_COTROL
      OR      D5000.1  ; CKT2_AUTO_COTROL
      ANB
      AND     T854  ; NST5_MACHINE_PALLET_EMPTY_TIMR
      SET     D8040.7  ; NST5_MACHINE_STOP_GATE_CYCL_CMPL
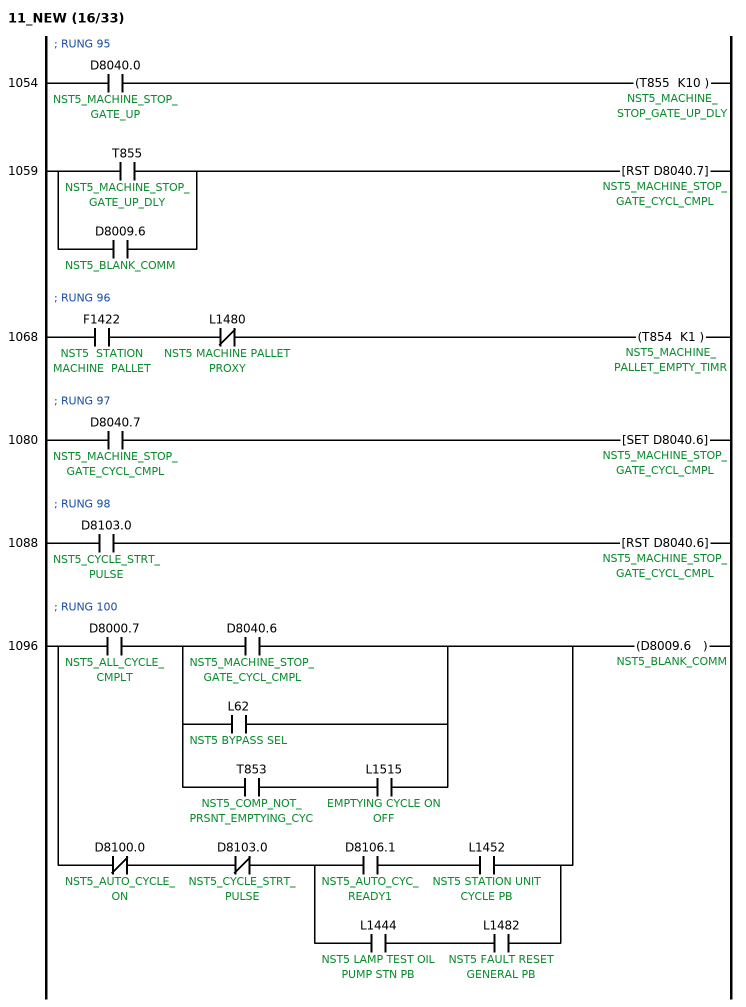
; RUNG 95
1054  LD      D8040.0  ; NST5_MACHINE_STOP_GATE_UP
      OUT     T855 K10  ; NST5_MACHINE_STOP_GATE_UP_DLY
1059  LD      T855  ; NST5_MACHINE_STOP_GATE_UP_DLY
      OR      D8009.6  ; NST5_BLANK_COMM
      RST     D8040.7  ; NST5_MACHINE_STOP_GATE_CYCL_CMPL
; RUNG 96
1068  LD      F1422  ; NST5  STATION  MACHINE  PALLET
      ANI     L1480  ; NST5 MACHINE PALLET PROXY
      OUT     T854 K1  ; NST5_MACHINE_PALLET_EMPTY_TIMR
; RUNG 97
1080  LD      D8040.7  ; NST5_MACHINE_STOP_GATE_CYCL_CMPL
      SET     D8040.6  ; NST5_MACHINE_STOP_GATE_CYCL_CMPL
; RUNG 98
1088  LD      D8103.0  ; NST5_CYCLE_STRT_PULSE
      RST     D8040.6  ; NST5_MACHINE_STOP_GATE_CYCL_CMPL
; RUNG 100
1096  LD      D8000.7  ; NST5_ALL_CYCLE_CMPLT
      LD      D8040.6  ; NST5_MACHINE_STOP_GATE_CYCL_CMPL
      OR      L62  ; NST5 BYPASS SEL
      LD      T853  ; NST5_COMP_NOT_PRSNT_EMPTYING_CYC
      AND     L1515  ; EMPTYING CYCLE ON OFF
      ORB
      ANB
      LDI     D8100.0  ; NST5_AUTO_CYCLE_ON
      ANI     D8103.0  ; NST5_CYCLE_STRT_PULSE
      LD      D8106.1  ; NST5_AUTO_CYC_READY1
      AND     L1452  ; NST5 STATION UNIT CYCLE PB
      LD      L1444  ; NST5 LAMP TEST OIL PUMP STN PB
      AND     L1482  ; NST5 FAULT RESET GENERAL PB
      ORB
      ANB
      ORB
      OUT     D8009.6  ; NST5_BLANK_COMM
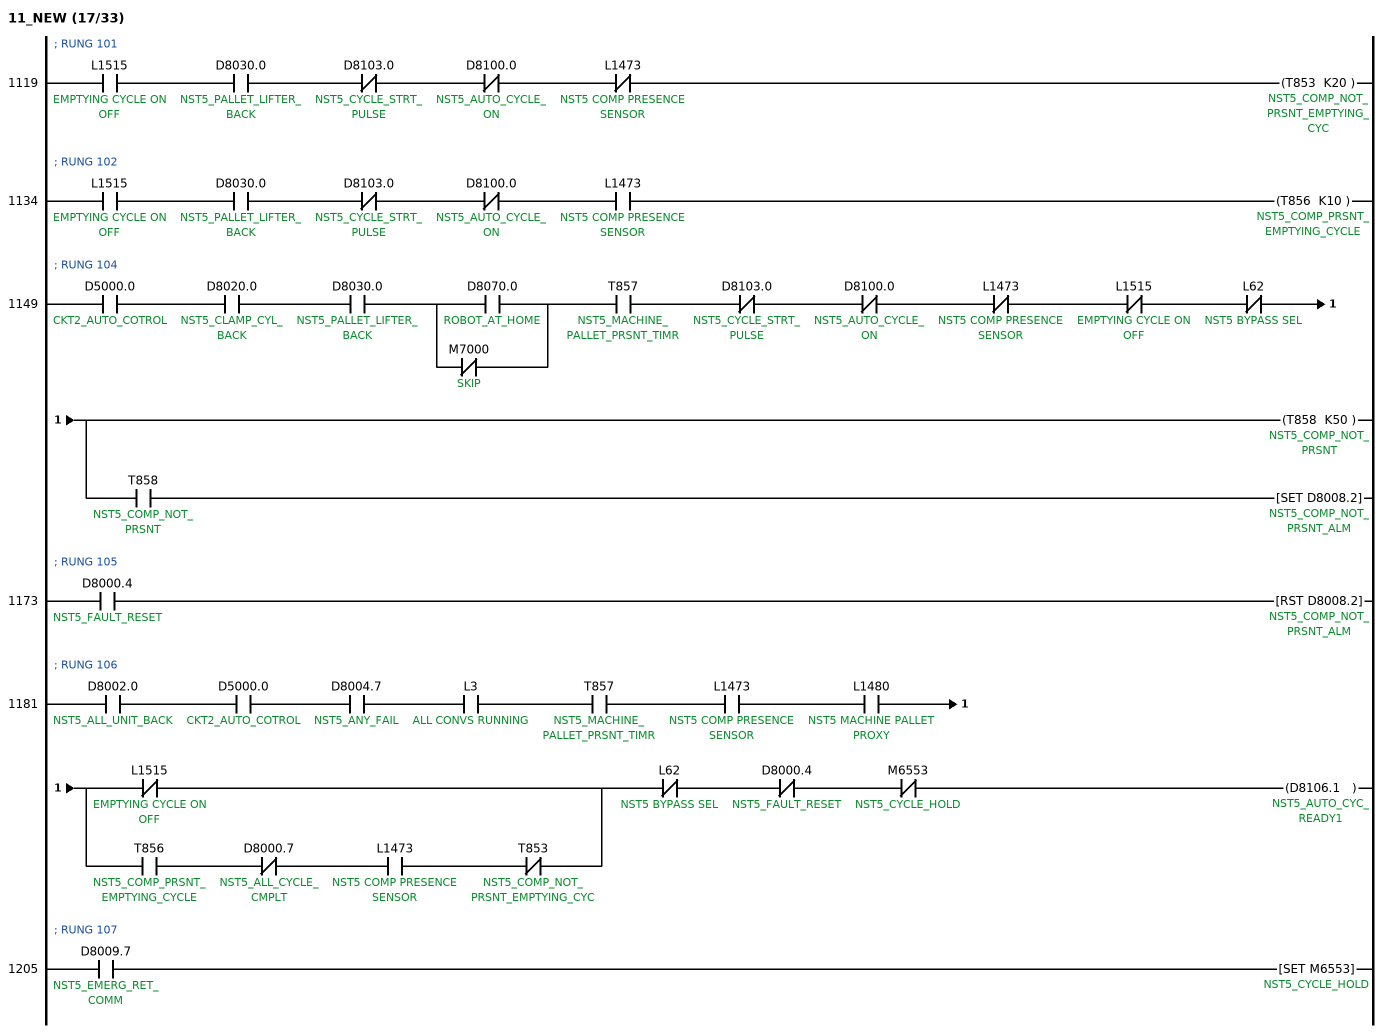
; RUNG 101
1119  LD      L1515  ; EMPTYING CYCLE ON OFF
      AND     D8030.0  ; NST5_PALLET_LIFTER_BACK
      ANI     D8103.0  ; NST5_CYCLE_STRT_PULSE
      ANI     D8100.0  ; NST5_AUTO_CYCLE_ON
      ANI     L1473  ; NST5 COMP PRESENCE SENSOR
      OUT     T853 K20  ; NST5_COMP_NOT_PRSNT_EMPTYING_CYC
; RUNG 102
1134  LD      L1515  ; EMPTYING CYCLE ON OFF
      AND     D8030.0  ; NST5_PALLET_LIFTER_BACK
      ANI     D8103.0  ; NST5_CYCLE_STRT_PULSE
      ANI     D8100.0  ; NST5_AUTO_CYCLE_ON
      AND     L1473  ; NST5 COMP PRESENCE SENSOR
      OUT     T856 K10  ; NST5_COMP_PRSNT_EMPTYING_CYCLE
; RUNG 104
1149  LD      D5000.0  ; CKT2_AUTO_COTROL
      AND     D8020.0  ; NST5_CLAMP_CYL_BACK
      AND     D8030.0  ; NST5_PALLET_LIFTER_BACK
      LD      D8070.0  ; ROBOT_AT_HOME
      ORI     M7000  ; SKIP
      ANB
      AND     T857  ; NST5_MACHINE_PALLET_PRSNT_TIMR
      ANI     D8103.0  ; NST5_CYCLE_STRT_PULSE
      ANI     D8100.0  ; NST5_AUTO_CYCLE_ON
      ANI     L1473  ; NST5 COMP PRESENCE SENSOR
      ANI     L1515  ; EMPTYING CYCLE ON OFF
      ANI     L62  ; NST5 BYPASS SEL
      OUT     T858 K50  ; NST5_COMP_NOT_PRSNT
      AND     T858  ; NST5_COMP_NOT_PRSNT
      SET     D8008.2  ; NST5_COMP_NOT_PRSNT_ALM
; RUNG 105
1173  LD      D8000.4  ; NST5_FAULT_RESET
      RST     D8008.2  ; NST5_COMP_NOT_PRSNT_ALM
; RUNG 106
1181  LD      D8002.0  ; NST5_ALL_UNIT_BACK
      AND     D5000.0  ; CKT2_AUTO_COTROL
      AND     D8004.7  ; NST5_ANY_FAIL
      AND     L3  ; ALL CONVS RUNNING
      AND     T857  ; NST5_MACHINE_PALLET_PRSNT_TIMR
      AND     L1473  ; NST5 COMP PRESENCE SENSOR
      AND     L1480  ; NST5 MACHINE PALLET PROXY
      LDI     L1515  ; EMPTYING CYCLE ON OFF
      LD      T856  ; NST5_COMP_PRSNT_EMPTYING_CYCLE
      ANI     D8000.7  ; NST5_ALL_CYCLE_CMPLT
      AND     L1473  ; NST5 COMP PRESENCE SENSOR
      ANI     T853  ; NST5_COMP_NOT_PRSNT_EMPTYING_CYC
      ORB
      ANB
      ANI     L62  ; NST5 BYPASS SEL
      ANI     D8000.4  ; NST5_FAULT_RESET
      ANI     M6553  ; NST5_CYCLE_HOLD
      OUT     D8106.1  ; NST5_AUTO_CYC_READY1
; RUNG 107
1205  LD      D8009.7  ; NST5_EMERG_RET_COMM
      SET     M6553  ; NST5_CYCLE_HOLD
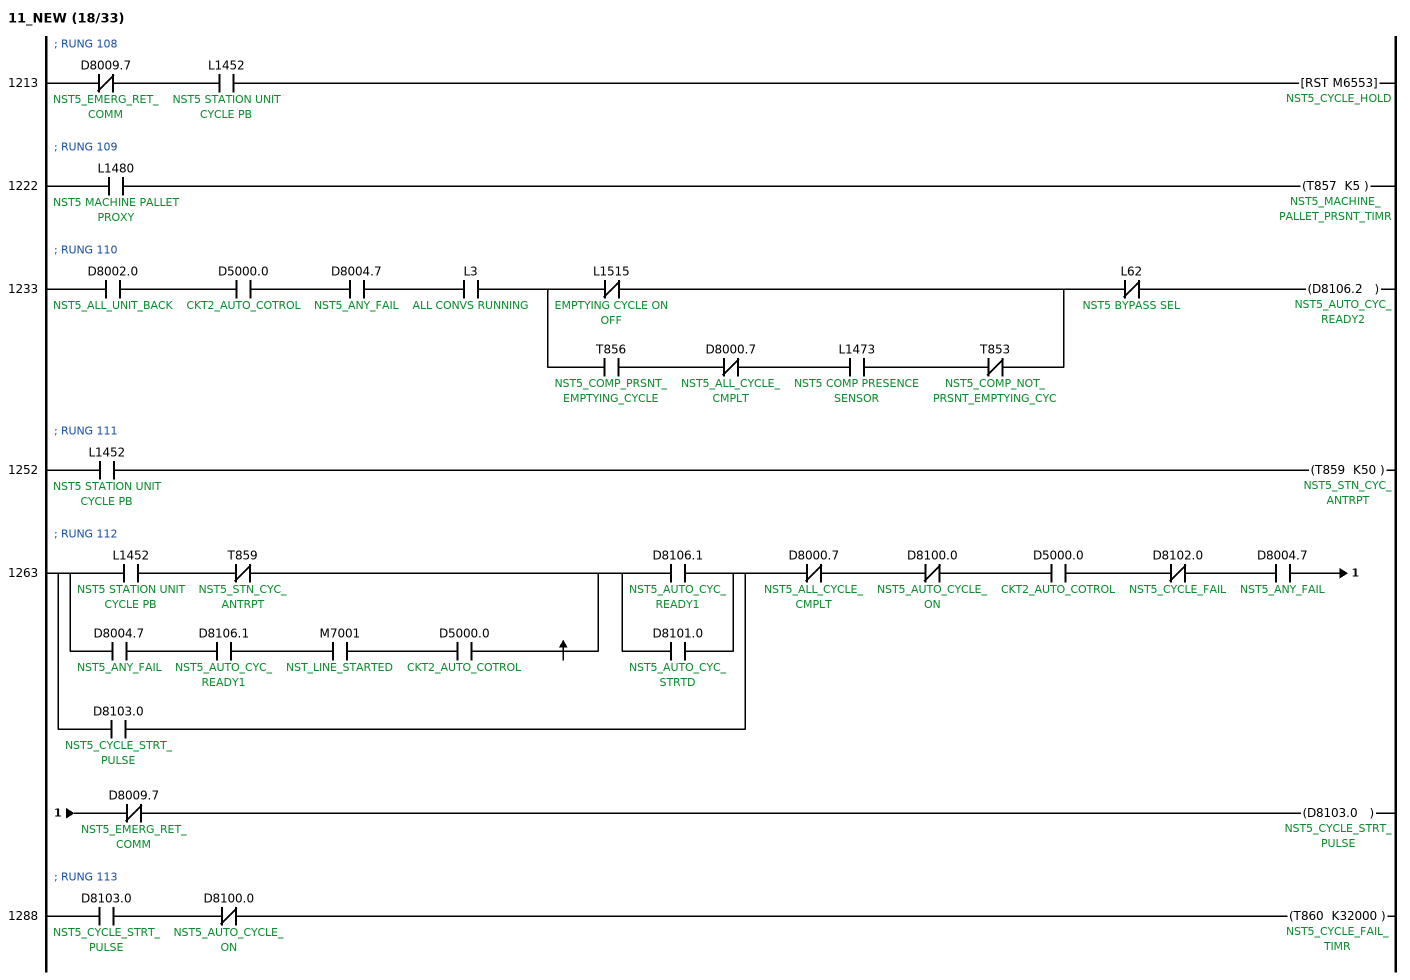
; RUNG 108
1213  LDI     D8009.7  ; NST5_EMERG_RET_COMM
      AND     L1452  ; NST5 STATION UNIT CYCLE PB
      RST     M6553  ; NST5_CYCLE_HOLD
; RUNG 109
1222  LD      L1480  ; NST5 MACHINE PALLET PROXY
      OUT     T857 K5  ; NST5_MACHINE_PALLET_PRSNT_TIMR
; RUNG 110
1233  LD      D8002.0  ; NST5_ALL_UNIT_BACK
      AND     D5000.0  ; CKT2_AUTO_COTROL
      AND     D8004.7  ; NST5_ANY_FAIL
      AND     L3  ; ALL CONVS RUNNING
      LDI     L1515  ; EMPTYING CYCLE ON OFF
      LD      T856  ; NST5_COMP_PRSNT_EMPTYING_CYCLE
      ANI     D8000.7  ; NST5_ALL_CYCLE_CMPLT
      AND     L1473  ; NST5 COMP PRESENCE SENSOR
      ANI     T853  ; NST5_COMP_NOT_PRSNT_EMPTYING_CYC
      ORB
      ANB
      ANI     L62  ; NST5 BYPASS SEL
      OUT     D8106.2  ; NST5_AUTO_CYC_READY2
; RUNG 111
1252  LD      L1452  ; NST5 STATION UNIT CYCLE PB
      OUT     T859 K50  ; NST5_STN_CYC_ANTRPT
; RUNG 112
1263  LD      L1452  ; NST5 STATION UNIT CYCLE PB
      ANI     T859  ; NST5_STN_CYC_ANTRPT
      LD      D8004.7  ; NST5_ANY_FAIL
      AND     D8106.1  ; NST5_AUTO_CYC_READY1
      AND     M7001  ; NST_LINE_STARTED
      AND     D5000.0  ; CKT2_AUTO_COTROL
      MEP
      ORB
      LD      D8106.1  ; NST5_AUTO_CYC_READY1
      OR      D8101.0  ; NST5_AUTO_CYC_STRTD
      ANB
      OR      D8103.0  ; NST5_CYCLE_STRT_PULSE
      ANI     D8000.7  ; NST5_ALL_CYCLE_CMPLT
      ANI     D8100.0  ; NST5_AUTO_CYCLE_ON
      AND     D5000.0  ; CKT2_AUTO_COTROL
      ANI     D8102.0  ; NST5_CYCLE_FAIL
      AND     D8004.7  ; NST5_ANY_FAIL
      ANI     D8009.7  ; NST5_EMERG_RET_COMM
      OUT     D8103.0  ; NST5_CYCLE_STRT_PULSE
; RUNG 113
1288  LD      D8103.0  ; NST5_CYCLE_STRT_PULSE
      ANI     D8100.0  ; NST5_AUTO_CYCLE_ON
      OUT     T860 K32000  ; NST5_CYCLE_FAIL_TIMR
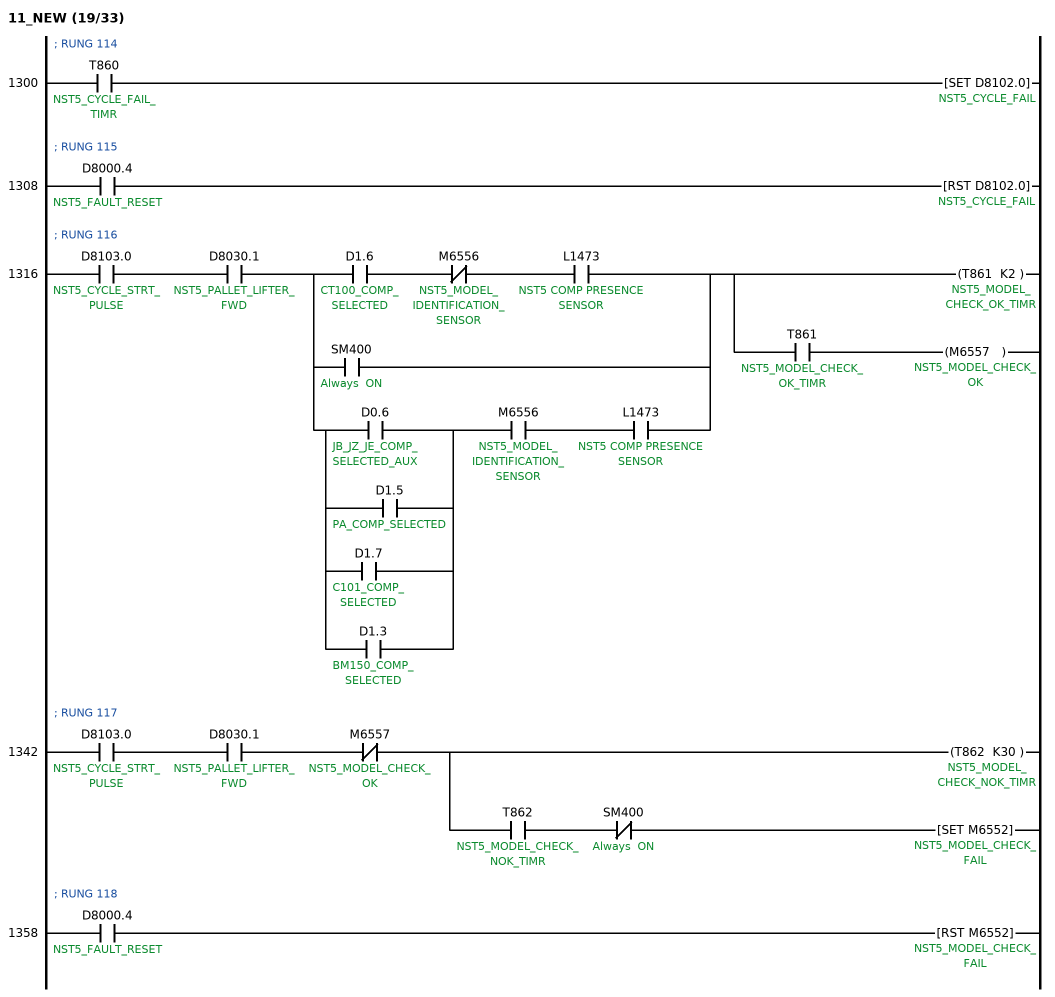
; RUNG 114
1300  LD      T860  ; NST5_CYCLE_FAIL_TIMR
      SET     D8102.0  ; NST5_CYCLE_FAIL
; RUNG 115
1308  LD      D8000.4  ; NST5_FAULT_RESET
      RST     D8102.0  ; NST5_CYCLE_FAIL
; RUNG 116
1316  LD      D8103.0  ; NST5_CYCLE_STRT_PULSE
      AND     D8030.1  ; NST5_PALLET_LIFTER_FWD
      LD      D1.6  ; CT100_COMP_SELECTED
      ANI     M6556  ; NST5_MODEL_IDENTIFICATION_SENSOR
      AND     L1473  ; NST5 COMP PRESENCE SENSOR
      OR      SM400  ; Always  ON
      LD      D0.6  ; JB_JZ_JE_COMP_SELECTED_AUX
      OR      D1.5  ; PA_COMP_SELECTED
      OR      D1.7  ; C101_COMP_SELECTED
      OR      D1.3  ; BM150_COMP_SELECTED
      AND     M6556  ; NST5_MODEL_IDENTIFICATION_SENSOR
      AND     L1473  ; NST5 COMP PRESENCE SENSOR
      ORB
      ANB
      OUT     T861 K2  ; NST5_MODEL_CHECK_OK_TIMR
      AND     T861  ; NST5_MODEL_CHECK_OK_TIMR
      OUT     M6557  ; NST5_MODEL_CHECK_OK
; RUNG 117
1342  LD      D8103.0  ; NST5_CYCLE_STRT_PULSE
      AND     D8030.1  ; NST5_PALLET_LIFTER_FWD
      ANI     M6557  ; NST5_MODEL_CHECK_OK
      OUT     T862 K30  ; NST5_MODEL_CHECK_NOK_TIMR
      AND     T862  ; NST5_MODEL_CHECK_NOK_TIMR
      ANI     SM400  ; Always  ON
      SET     M6552  ; NST5_MODEL_CHECK_FAIL
; RUNG 118
1358  LD      D8000.4  ; NST5_FAULT_RESET
      RST     M6552  ; NST5_MODEL_CHECK_FAIL
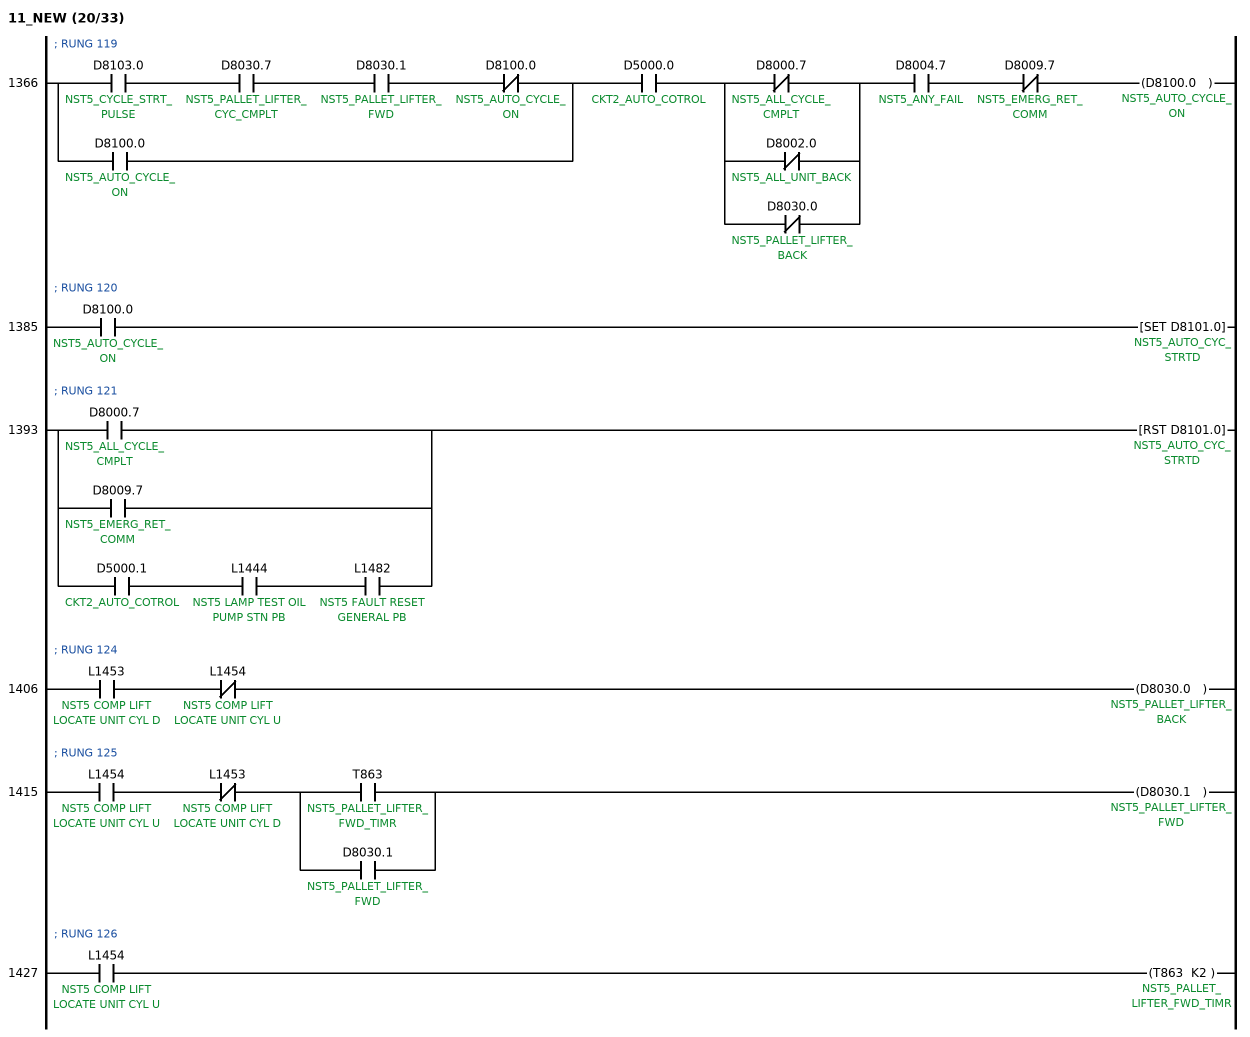
; RUNG 119
1366  LD      D8103.0  ; NST5_CYCLE_STRT_PULSE
      AND     D8030.7  ; NST5_PALLET_LIFTER_CYC_CMPLT
      AND     D8030.1  ; NST5_PALLET_LIFTER_FWD
      ANI     D8100.0  ; NST5_AUTO_CYCLE_ON
      OR      D8100.0  ; NST5_AUTO_CYCLE_ON
      AND     D5000.0  ; CKT2_AUTO_COTROL
      LDI     D8000.7  ; NST5_ALL_CYCLE_CMPLT
      ORI     D8002.0  ; NST5_ALL_UNIT_BACK
      ORI     D8030.0  ; NST5_PALLET_LIFTER_BACK
      ANB
      AND     D8004.7  ; NST5_ANY_FAIL
      ANI     D8009.7  ; NST5_EMERG_RET_COMM
      OUT     D8100.0  ; NST5_AUTO_CYCLE_ON
; RUNG 120
1385  LD      D8100.0  ; NST5_AUTO_CYCLE_ON
      SET     D8101.0  ; NST5_AUTO_CYC_STRTD
; RUNG 121
1393  LD      D8000.7  ; NST5_ALL_CYCLE_CMPLT
      OR      D8009.7  ; NST5_EMERG_RET_COMM
      LD      D5000.1  ; CKT2_AUTO_COTROL
      AND     L1444  ; NST5 LAMP TEST OIL PUMP STN PB
      AND     L1482  ; NST5 FAULT RESET GENERAL PB
      ORB
      RST     D8101.0  ; NST5_AUTO_CYC_STRTD
; RUNG 124
1406  LD      L1453  ; NST5 COMP LIFT LOCATE UNIT CYL D
      ANI     L1454  ; NST5 COMP LIFT LOCATE UNIT CYL U
      OUT     D8030.0  ; NST5_PALLET_LIFTER_BACK
; RUNG 125
1415  LD      L1454  ; NST5 COMP LIFT LOCATE UNIT CYL U
      ANI     L1453  ; NST5 COMP LIFT LOCATE UNIT CYL D
      LD      T863  ; NST5_PALLET_LIFTER_FWD_TIMR
      OR      D8030.1  ; NST5_PALLET_LIFTER_FWD
      ANB
      OUT     D8030.1  ; NST5_PALLET_LIFTER_FWD
; RUNG 126
1427  LD      L1454  ; NST5 COMP LIFT LOCATE UNIT CYL U
      OUT     T863 K2  ; NST5_PALLET_LIFTER_FWD_TIMR
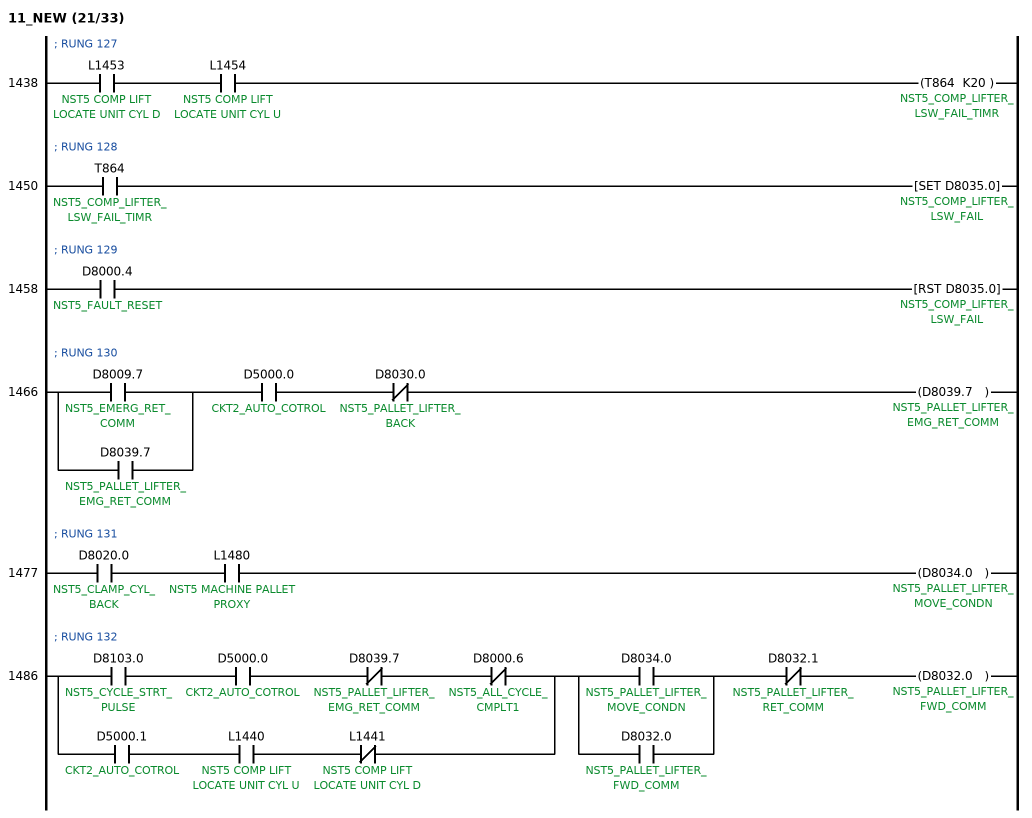
; RUNG 127
1438  LD      L1453  ; NST5 COMP LIFT LOCATE UNIT CYL D
      AND     L1454  ; NST5 COMP LIFT LOCATE UNIT CYL U
      OUT     T864 K20  ; NST5_COMP_LIFTER_LSW_FAIL_TIMR
; RUNG 128
1450  LD      T864  ; NST5_COMP_LIFTER_LSW_FAIL_TIMR
      SET     D8035.0  ; NST5_COMP_LIFTER_LSW_FAIL
; RUNG 129
1458  LD      D8000.4  ; NST5_FAULT_RESET
      RST     D8035.0  ; NST5_COMP_LIFTER_LSW_FAIL
; RUNG 130
1466  LD      D8009.7  ; NST5_EMERG_RET_COMM
      OR      D8039.7  ; NST5_PALLET_LIFTER_EMG_RET_COMM
      AND     D5000.0  ; CKT2_AUTO_COTROL
      ANI     D8030.0  ; NST5_PALLET_LIFTER_BACK
      OUT     D8039.7  ; NST5_PALLET_LIFTER_EMG_RET_COMM
; RUNG 131
1477  LD      D8020.0  ; NST5_CLAMP_CYL_BACK
      AND     L1480  ; NST5 MACHINE PALLET PROXY
      OUT     D8034.0  ; NST5_PALLET_LIFTER_MOVE_CONDN
; RUNG 132
1486  LD      D8103.0  ; NST5_CYCLE_STRT_PULSE
      AND     D5000.0  ; CKT2_AUTO_COTROL
      ANI     D8039.7  ; NST5_PALLET_LIFTER_EMG_RET_COMM
      ANI     D8000.6  ; NST5_ALL_CYCLE_CMPLT1
      LD      D5000.1  ; CKT2_AUTO_COTROL
      AND     L1440  ; NST5 COMP LIFT LOCATE UNIT CYL U
      ANI     L1441  ; NST5 COMP LIFT LOCATE UNIT CYL D
      ORB
      LD      D8034.0  ; NST5_PALLET_LIFTER_MOVE_CONDN
      OR      D8032.0  ; NST5_PALLET_LIFTER_FWD_COMM
      ANB
      ANI     D8032.1  ; NST5_PALLET_LIFTER_RET_COMM
      OUT     D8032.0  ; NST5_PALLET_LIFTER_FWD_COMM
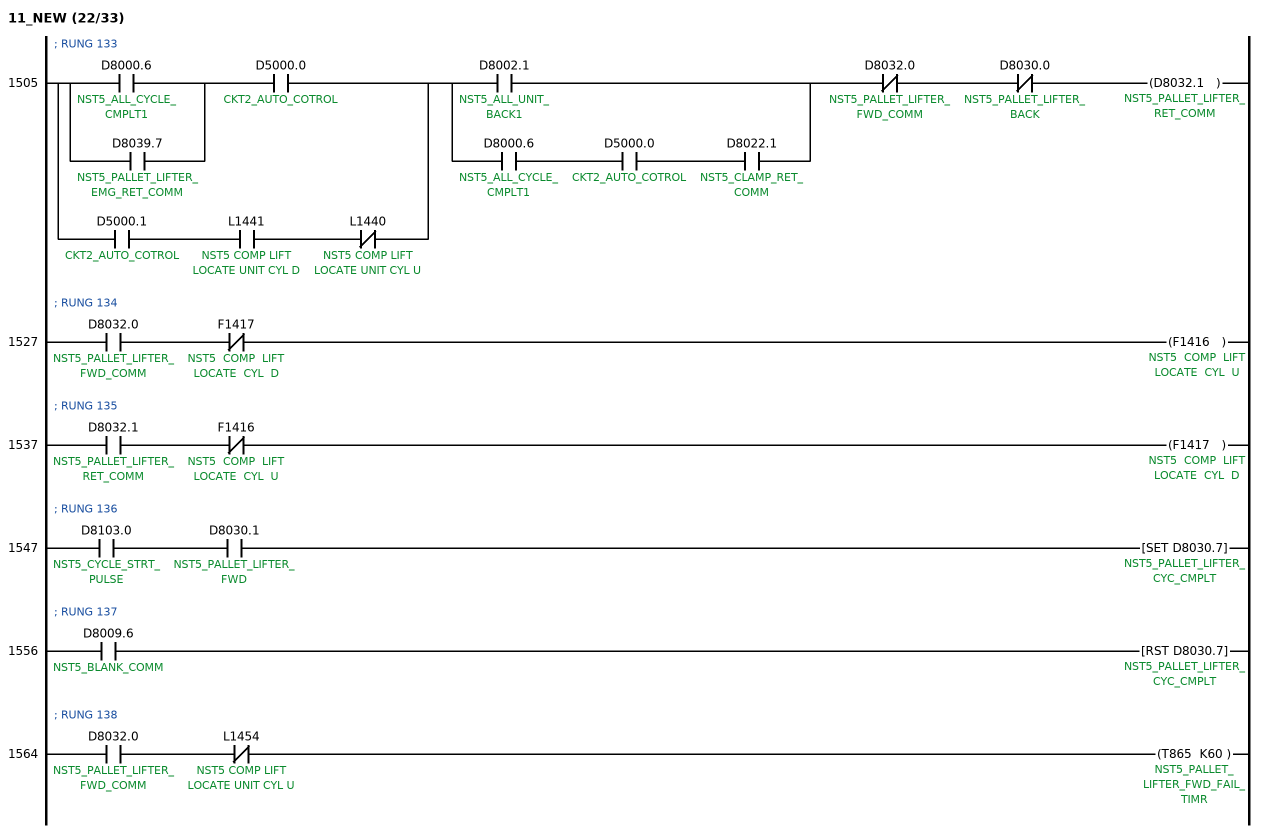
; RUNG 133
1505  LD      D8000.6  ; NST5_ALL_CYCLE_CMPLT1
      OR      D8039.7  ; NST5_PALLET_LIFTER_EMG_RET_COMM
      AND     D5000.0  ; CKT2_AUTO_COTROL
      LD      D5000.1  ; CKT2_AUTO_COTROL
      AND     L1441  ; NST5 COMP LIFT LOCATE UNIT CYL D
      ANI     L1440  ; NST5 COMP LIFT LOCATE UNIT CYL U
      ORB
      LD      D8002.1  ; NST5_ALL_UNIT_BACK1
      LD      D8000.6  ; NST5_ALL_CYCLE_CMPLT1
      AND     D5000.0  ; CKT2_AUTO_COTROL
      AND     D8022.1  ; NST5_CLAMP_RET_COMM
      ORB
      ANB
      ANI     D8032.0  ; NST5_PALLET_LIFTER_FWD_COMM
      ANI     D8030.0  ; NST5_PALLET_LIFTER_BACK
      OUT     D8032.1  ; NST5_PALLET_LIFTER_RET_COMM
; RUNG 134
1527  LD      D8032.0  ; NST5_PALLET_LIFTER_FWD_COMM
      ANI     F1417  ; NST5  COMP  LIFT  LOCATE  CYL  D
      OUT     F1416  ; NST5  COMP  LIFT  LOCATE  CYL  U
; RUNG 135
1537  LD      D8032.1  ; NST5_PALLET_LIFTER_RET_COMM
      ANI     F1416  ; NST5  COMP  LIFT  LOCATE  CYL  U
      OUT     F1417  ; NST5  COMP  LIFT  LOCATE  CYL  D
; RUNG 136
1547  LD      D8103.0  ; NST5_CYCLE_STRT_PULSE
      AND     D8030.1  ; NST5_PALLET_LIFTER_FWD
      SET     D8030.7  ; NST5_PALLET_LIFTER_CYC_CMPLT
; RUNG 137
1556  LD      D8009.6  ; NST5_BLANK_COMM
      RST     D8030.7  ; NST5_PALLET_LIFTER_CYC_CMPLT
; RUNG 138
1564  LD      D8032.0  ; NST5_PALLET_LIFTER_FWD_COMM
      ANI     L1454  ; NST5 COMP LIFT LOCATE UNIT CYL U
      OUT     T865 K60  ; NST5_PALLET_LIFTER_FWD_FAIL_TIMR
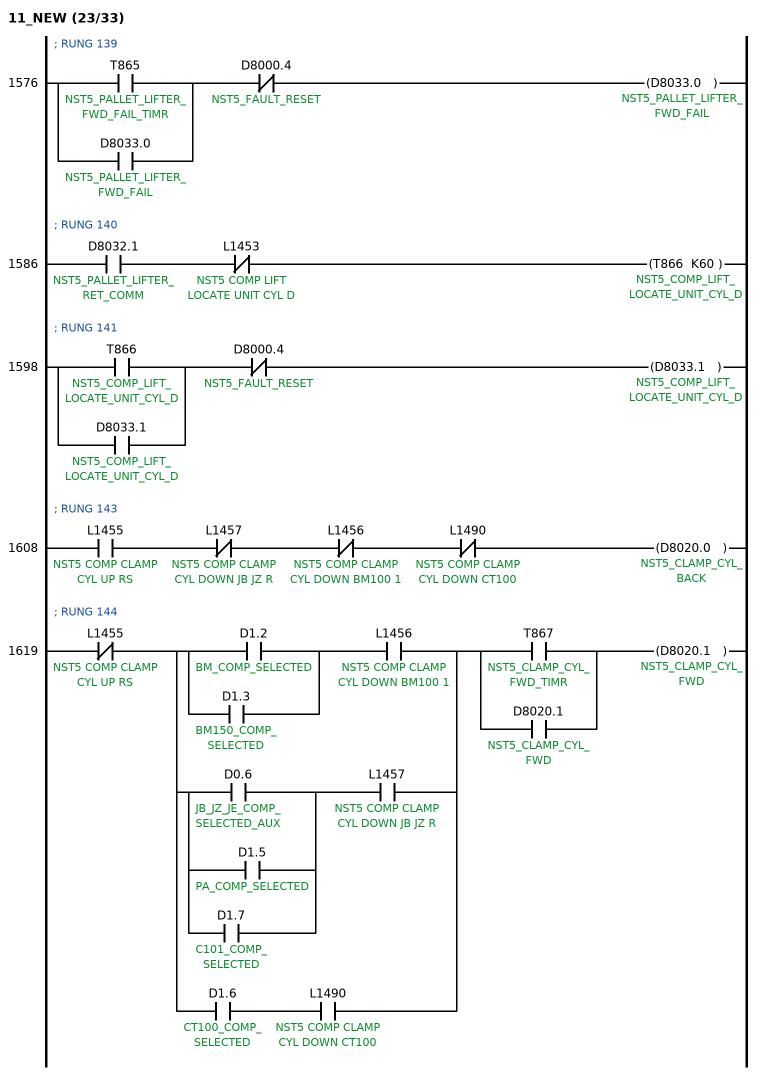
; RUNG 139
1576  LD      T865  ; NST5_PALLET_LIFTER_FWD_FAIL_TIMR
      OR      D8033.0  ; NST5_PALLET_LIFTER_FWD_FAIL
      ANI     D8000.4  ; NST5_FAULT_RESET
      OUT     D8033.0  ; NST5_PALLET_LIFTER_FWD_FAIL
; RUNG 140
1586  LD      D8032.1  ; NST5_PALLET_LIFTER_RET_COMM
      ANI     L1453  ; NST5 COMP LIFT LOCATE UNIT CYL D
      OUT     T866 K60  ; NST5_COMP_LIFT_LOCATE_UNIT_CYL_D
; RUNG 141
1598  LD      T866  ; NST5_COMP_LIFT_LOCATE_UNIT_CYL_D
      OR      D8033.1  ; NST5_COMP_LIFT_LOCATE_UNIT_CYL_D
      ANI     D8000.4  ; NST5_FAULT_RESET
      OUT     D8033.1  ; NST5_COMP_LIFT_LOCATE_UNIT_CYL_D
; RUNG 143
1608  LD      L1455  ; NST5 COMP CLAMP CYL UP RS
      ANI     L1457  ; NST5 COMP CLAMP CYL DOWN JB JZ R
      ANI     L1456  ; NST5 COMP CLAMP CYL DOWN BM100 1
      ANI     L1490  ; NST5 COMP CLAMP CYL DOWN CT100
      OUT     D8020.0  ; NST5_CLAMP_CYL_BACK
; RUNG 144
1619  LDI     L1455  ; NST5 COMP CLAMP CYL UP RS
      LD      D1.2  ; BM_COMP_SELECTED
      OR      D1.3  ; BM150_COMP_SELECTED
      AND     L1456  ; NST5 COMP CLAMP CYL DOWN BM100 1
      LD      D0.6  ; JB_JZ_JE_COMP_SELECTED_AUX
      OR      D1.5  ; PA_COMP_SELECTED
      OR      D1.7  ; C101_COMP_SELECTED
      AND     L1457  ; NST5 COMP CLAMP CYL DOWN JB JZ R
      ORB
      LD      D1.6  ; CT100_COMP_SELECTED
      AND     L1490  ; NST5 COMP CLAMP CYL DOWN CT100
      ORB
      ANB
      LD      T867  ; NST5_CLAMP_CYL_FWD_TIMR
      OR      D8020.1  ; NST5_CLAMP_CYL_FWD
      ANB
      OUT     D8020.1  ; NST5_CLAMP_CYL_FWD
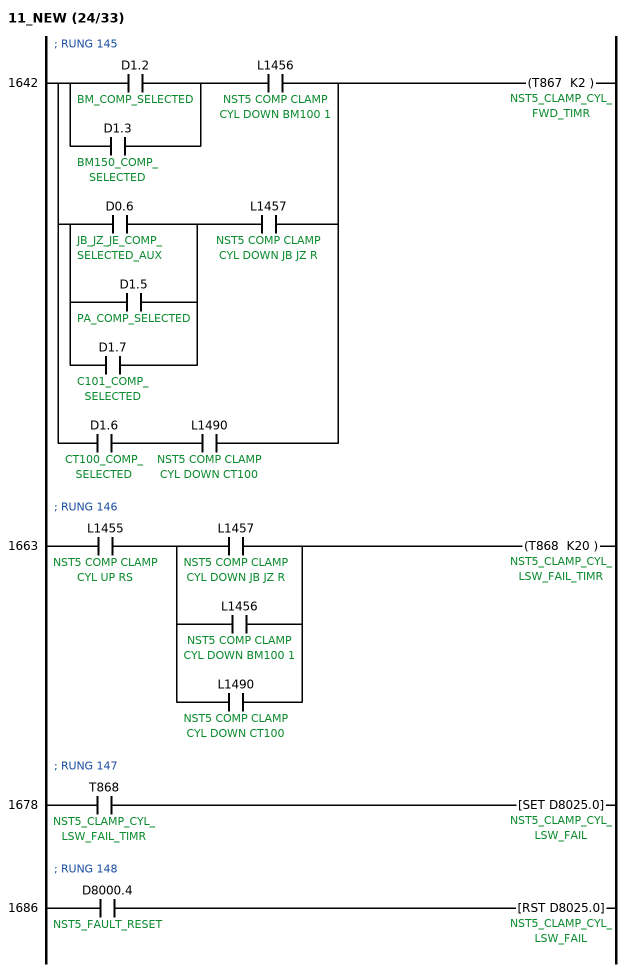
; RUNG 145
1642  LD      D1.2  ; BM_COMP_SELECTED
      OR      D1.3  ; BM150_COMP_SELECTED
      AND     L1456  ; NST5 COMP CLAMP CYL DOWN BM100 1
      LD      D0.6  ; JB_JZ_JE_COMP_SELECTED_AUX
      OR      D1.5  ; PA_COMP_SELECTED
      OR      D1.7  ; C101_COMP_SELECTED
      AND     L1457  ; NST5 COMP CLAMP CYL DOWN JB JZ R
      ORB
      LD      D1.6  ; CT100_COMP_SELECTED
      AND     L1490  ; NST5 COMP CLAMP CYL DOWN CT100
      ORB
      OUT     T867 K2  ; NST5_CLAMP_CYL_FWD_TIMR
; RUNG 146
1663  LD      L1455  ; NST5 COMP CLAMP CYL UP RS
      LD      L1457  ; NST5 COMP CLAMP CYL DOWN JB JZ R
      OR      L1456  ; NST5 COMP CLAMP CYL DOWN BM100 1
      OR      L1490  ; NST5 COMP CLAMP CYL DOWN CT100
      ANB
      OUT     T868 K20  ; NST5_CLAMP_CYL_LSW_FAIL_TIMR
; RUNG 147
1678  LD      T868  ; NST5_CLAMP_CYL_LSW_FAIL_TIMR
      SET     D8025.0  ; NST5_CLAMP_CYL_LSW_FAIL
; RUNG 148
1686  LD      D8000.4  ; NST5_FAULT_RESET
      RST     D8025.0  ; NST5_CLAMP_CYL_LSW_FAIL
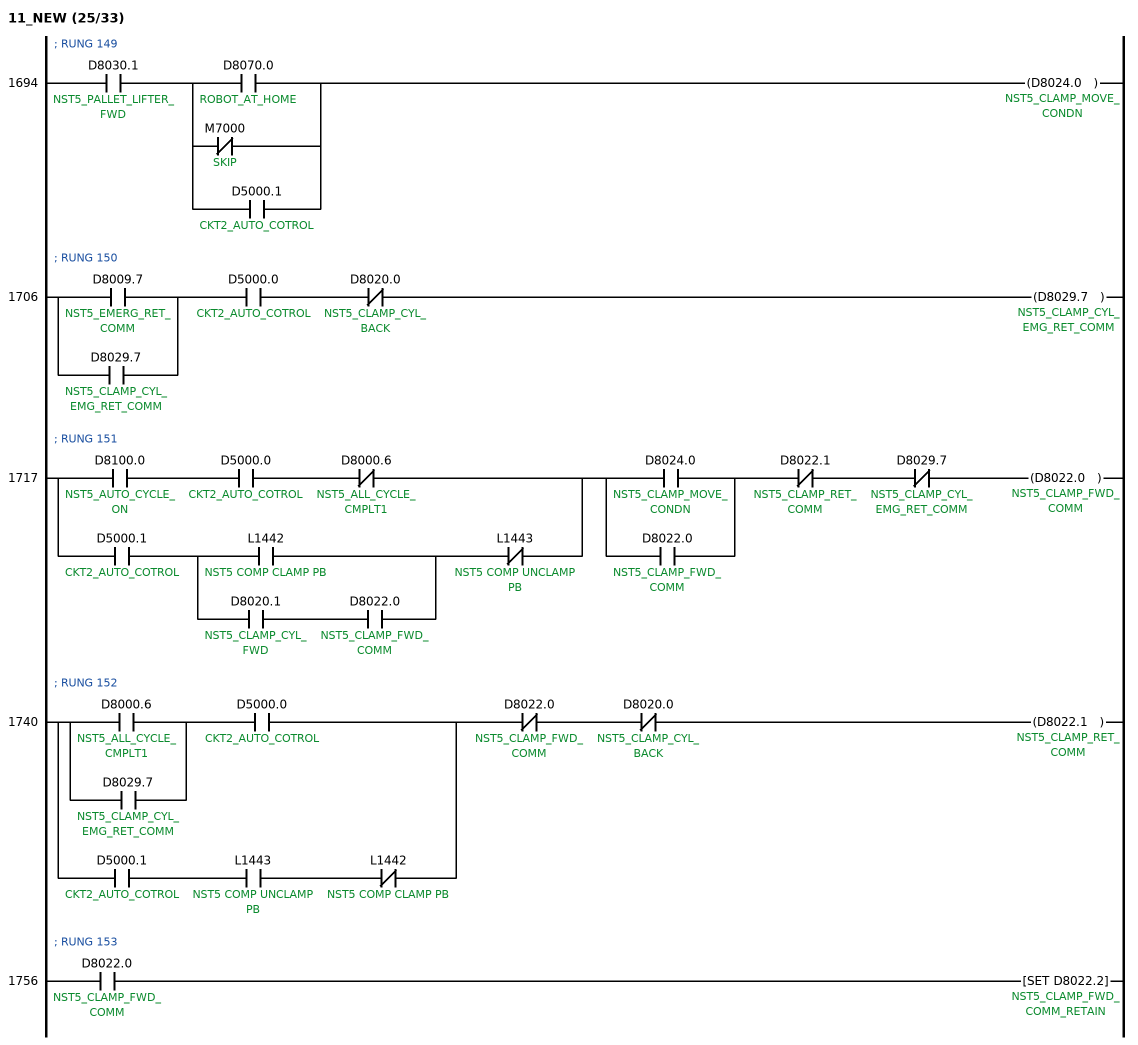
; RUNG 149
1694  LD      D8030.1  ; NST5_PALLET_LIFTER_FWD
      LD      D8070.0  ; ROBOT_AT_HOME
      ORI     M7000  ; SKIP
      OR      D5000.1  ; CKT2_AUTO_COTROL
      ANB
      OUT     D8024.0  ; NST5_CLAMP_MOVE_CONDN
; RUNG 150
1706  LD      D8009.7  ; NST5_EMERG_RET_COMM
      OR      D8029.7  ; NST5_CLAMP_CYL_EMG_RET_COMM
      AND     D5000.0  ; CKT2_AUTO_COTROL
      ANI     D8020.0  ; NST5_CLAMP_CYL_BACK
      OUT     D8029.7  ; NST5_CLAMP_CYL_EMG_RET_COMM
; RUNG 151
1717  LD      D8100.0  ; NST5_AUTO_CYCLE_ON
      AND     D5000.0  ; CKT2_AUTO_COTROL
      ANI     D8000.6  ; NST5_ALL_CYCLE_CMPLT1
      LD      D5000.1  ; CKT2_AUTO_COTROL
      LD      L1442  ; NST5 COMP CLAMP PB
      LD      D8020.1  ; NST5_CLAMP_CYL_FWD
      AND     D8022.0  ; NST5_CLAMP_FWD_COMM
      ORB
      ANB
      ANI     L1443  ; NST5 COMP UNCLAMP PB
      ORB
      LD      D8024.0  ; NST5_CLAMP_MOVE_CONDN
      OR      D8022.0  ; NST5_CLAMP_FWD_COMM
      ANB
      ANI     D8022.1  ; NST5_CLAMP_RET_COMM
      ANI     D8029.7  ; NST5_CLAMP_CYL_EMG_RET_COMM
      OUT     D8022.0  ; NST5_CLAMP_FWD_COMM
; RUNG 152
1740  LD      D8000.6  ; NST5_ALL_CYCLE_CMPLT1
      OR      D8029.7  ; NST5_CLAMP_CYL_EMG_RET_COMM
      AND     D5000.0  ; CKT2_AUTO_COTROL
      LD      D5000.1  ; CKT2_AUTO_COTROL
      AND     L1443  ; NST5 COMP UNCLAMP PB
      ANI     L1442  ; NST5 COMP CLAMP PB
      ORB
      ANI     D8022.0  ; NST5_CLAMP_FWD_COMM
      ANI     D8020.0  ; NST5_CLAMP_CYL_BACK
      OUT     D8022.1  ; NST5_CLAMP_RET_COMM
; RUNG 153
1756  LD      D8022.0  ; NST5_CLAMP_FWD_COMM
      SET     D8022.2  ; NST5_CLAMP_FWD_COMM_RETAIN
